// TwinCAT 3 PLC project PLC
// ProgramVersion: 3.1.4026.16
// libraries:
//   Tc2_ModbusRTU, * (Beckhoff Automation GmbH)
//   Tc2_Standard, * (Beckhoff Automation GmbH)
//   Tc2_SUPS, * (Beckhoff Automation GmbH)
//   Tc2_System, * (Beckhoff Automation GmbH)
//   Tc2_Utilities, * (Beckhoff Automation GmbH)
//   Tc3_Database, * (Beckhoff Automation GmbH)
//   Tc3_EventLogger, * (Beckhoff Automation GmbH)
// project tree:
//   DUTs/Database/ ST_AuditTrail.TcDUT, ST_BatchData.TcDUT, ST_OperatorAct.TcDUT, ST_ProcessData.TcDUT
//   DUTs/ EN_BatchEvents.TcDUT, EN_RecipeType.TcDUT, ST_Alarm.TcDUT, ST_Batch.TcDUT, ST_Control.TcDUT, ST_Diagnostic.TcDUT, ST_HMI.TcDUT, ST_HMI_Time.TcDUT, ST_LastBatch.TcDUT, ST_OPC.TcDUT, ST_ProcessCmd.TcDUT, ST_PythonHandshake.TcDUT, ST_RecipeList.TcDUT, ST_Report.TcDUT, ST_RX_Python.TcDUT, ST_Settings.TcDUT, ST_Time.TcDUT, ST_ToHMI.TcDUT, ST_TONP.TcDUT, ST_TX_Python.TcDUT
//   DUTs/Recipe/ ST_Cleaning_Phases.TcDUT, ST_Production_Phases.TcDUT, ST_Recipe_Production.TcDUT, ST_RecipeInfo.TcDUT, ST_Recipe_Cleaning.TcDUT
//   DUTs/ST_HMI/ ST_AlarmControl.TcDUT, ST_AuditControl.TcDUT, ST_BatchControl.TcDUT, ST_MachineControl.TcDUT, ST_ProcessControl.TcDUT, ST_RecipeControl.TcDUT, ST_ReportControl.TcDUT
//   DUTs/ST_ToHMI/ ST_Devices.TcDUT, ST_EnableControls.TcDUT, ST_Pipes.TcDUT, ST_ProcessVar.TcDUT, ST_Status.TcDUT
//   FB/Database/ FB_WriteChange.TcPOU, FB_WriteChange_STR.TcPOU, FB_WriteClick.TcPOU, FB_WriteEvent.TcPOU
//   FB/ FB_AnalogOutput.TcPOU, FB_AVG200.TcPOU, FB_Batch.TcPOU, FB_BatchLog.TcPOU, FB_Chopper_Ctrl.TcPOU, FB_Coil_Ctrl.TcPOU, FB_DeleteOldestFile.TcPOU, FB_FileSaveAs.TcPOU, FB_FileSaveAs_V02.TcPOU, FB_Mixer_Ctrl.TcPOU, FB_PythonScript.TcPOU, FB_Scale.TcPOU, FB_SystemDateTime.TcPOU, FB_TimeElapsed_HMI.TcPOU, FB_TONP.TcPOU, FB_Valve53_Ctrl.TcPOU, FB_Valve_Ctrl.TcPOU, F_Interlocks.TcPOU, F_OperationalTime.TcPOU, F_StepCMP.TcPOU, F_TimeBarHMI.TcPOU, F_TimerHMI.TcPOU
//   GVLs/ CONST.TcGVL, GV.TcGVL, IN.TcGVL, OUT.TcGVL, Recipes.TcGVL
//   Mapping/ ST_EL1819.TcDUT, ST_EL2809.TcDUT, ST_EL3174.TcDUT, ST_EL3214.TcDUT, ST_EL4008.TcDUT, ST_EL4124.TcDUT, ST_EL6021.TcDUT, ST_EL9110.TcDUT
//   / PlcTask.TcTTO
//   POUs/1. Main Control/ P1_00_MAIN.TcPOU, P1_01_Recipe.TcPOU, P1_02_Batch.TcPOU, P1_04_MachineControl.TcPOU, P1_03_Alarms.TcPOU
//   POUs/2. Process/Cleaning/ _Blowing.TcPOU, _Control.TcPOU, _Draining.TcPOU, _MainClean.TcPOU, _Mounting.TcPOU, _PreWash.TcPOU
//   POUs/2. Process/ P2_00_MAIN.TcPOU, P2_01_Production_Seq.TcPOU, P2_02_Cleaning_Seq.TcPOU, P2_03_Production_Ctrl.TcPOU, P2_04_Cleaning_Ctrl.TcPOU, P2_05_Process_Ctrl.TcPOU, P2_06_Device_Ctrl.TcPOU, _Chopper.TcPOU, _Mixer.TcPOU
//   POUs/2. Process/Production/ _Discharging.TcPOU, _Feeding.TcPOU, _Mixing.TcPOU
//   POUs/3. Report/ P3_00_MAIN.TcPOU, P3_01_BatchData.TcPOU, P3_03_ProcessData.TcPOU, P3_04_Alarms.TcPOU, P3_06_CreateReport.TcPOU, P3_07_SendReport.TcPOU, P3_08_OpenReport.TcPOU
//   POUs/4. Audit Trail/ P4_00_MAIN.TcPOU, P4_01_Write.TcPOU, P4_02_Read.TcPOU, P4_03_Export.TcPOU, P4_04_Delete.TcPOU, P4_05_DIskSize.TcPOU, P4_05_Send.TcPOU
//   POUs/5. HMI/ P5_00_MAIN.TcPOU, P5_01_EnableControls.TcPOU, P5_02_DiagramVisualisation.TcPOU, P5_03_OtherControl.TcPOU, P5_04_BatchStatus.TcPOU, P5_05_Screenshot.TcPOU, P5_06_Trends.TcPOU
//   POUs/ MAIN.TcPOU, P00_Mapping.TcPOU, P01_AnalogScaling.TcPOU, P02_GlobalSystemTime.TcPOU
// real-time tasks:
//   TASK PlcTask: cycle T#10ms, priority 20, ADS port 350
// I/O:
//   DEVICE PLC-ECAT (disabled), AmsNetId 169.254.227.12.5.1
//     BUS-ETCAT [EK1100 EtherCAT Coupler (2A E-Bus)]
//       PT100 (EL3214) (EL3214) [EL3214 4Ch. Ana. Input PT100 (RTD)]
//       Analog Input #1 (EL3174) [EL3174 4Ch. Ana. Input +/-10V Diff., +/-20mA SingleEnded, 16 Bit]
//       Analog Input #2 (EL3174) [EL3174 4Ch. Ana. Input +/-10V Diff., +/-20mA SingleEnded, 16 Bit]
//       Digital Input #1 (EL1819) [EL1819 16Ch. Dig. Input 24V, 10µs]
//       Analog Output #1 (EL4008) [EL4008 8Ch. Ana. Output 0-10V, 12bit]
//       Power Supply (EL9110) [EL9110 Power Supplier with LED (24V, Diagnostics)]
//       Digital Output #1 (EL2809) [EL2809 16Ch. Dig. Output 24V, 0.5A]
//       Digital Output #2 (EL2809) [EL2809 16Ch. Dig. Output 24V, 0.5A]
//       Modbus (EL6021) [EL6021 Interface (RS422/485)]
//       Term 9 (EL9011) [EL9011 End Terminal]
// variable links:
//   (this object) <-> PLC-ECAT/BUS-ETCAT/Analog Input #1 (EL3174)
//     PlcTask Inputs/P00_Mapping.AI1.Ch1_Error <-> AI Standard Channel 1/Status/Error
//     PlcTask Inputs/P00_Mapping.AI1.Ch2_Error <-> AI Standard Channel 2/Status/Error
//     PlcTask Inputs/P00_Mapping.AI1.Ch3_Error <-> AI Standard Channel 3/Status/Error
//     PlcTask Inputs/P00_Mapping.AI1.Ch4_Error <-> AI Standard Channel 4/Status/Error
//     PlcTask Inputs/P00_Mapping.AI1.Ch1_Value <-> AI Standard Channel 1/Value
//     PlcTask Inputs/P00_Mapping.AI1.Ch2_Value <-> AI Standard Channel 2/Value
//     PlcTask Inputs/P00_Mapping.AI1.Ch3_Value <-> AI Standard Channel 3/Value
//     PlcTask Inputs/P00_Mapping.AI1.Ch4_Value <-> AI Standard Channel 4/Value
//     PlcTask Inputs/P00_Mapping.AI1.State <-> InfoData/State
//   (this object) <-> PLC-ECAT/BUS-ETCAT/Analog Input #2 (EL3174)
//     PlcTask Inputs/P00_Mapping.AI2.Ch1_Error <-> AI Standard Channel 1/Status/Error
//     PlcTask Inputs/P00_Mapping.AI2.Ch2_Error <-> AI Standard Channel 2/Status/Error
//     PlcTask Inputs/P00_Mapping.AI2.Ch3_Error <-> AI Standard Channel 3/Status/Error
//     PlcTask Inputs/P00_Mapping.AI2.Ch4_Error <-> AI Standard Channel 4/Status/Error
//     PlcTask Inputs/P00_Mapping.AI2.Ch1_Value <-> AI Standard Channel 1/Value
//     PlcTask Inputs/P00_Mapping.AI2.Ch2_Value <-> AI Standard Channel 2/Value
//     PlcTask Inputs/P00_Mapping.AI2.Ch3_Value <-> AI Standard Channel 3/Value
//     PlcTask Inputs/P00_Mapping.AI2.Ch4_Value <-> AI Standard Channel 4/Value
//     PlcTask Inputs/P00_Mapping.AI2.State <-> InfoData/State
//   (this object) <-> PLC-ECAT/BUS-ETCAT/Analog Output #1 (EL4008)
//     PlcTask Inputs/P00_Mapping.AO1.State <-> InfoData/State
//     PlcTask Outputs/P00_Mapping.AO1.Ch1_Value <-> AO Outputs Channel 1/Analog output
//     PlcTask Outputs/P00_Mapping.AO1.Ch2_Value <-> AO Outputs Channel 2/Analog output
//     PlcTask Outputs/P00_Mapping.AO1.Ch3_Value <-> AO Outputs Channel 3/Analog output
//     PlcTask Outputs/P00_Mapping.AO1.Ch4_Value <-> AO Outputs Channel 4/Analog output
//   (this object) <-> PLC-ECAT/BUS-ETCAT/Digital Input #1 (EL1819)
//     PlcTask Inputs/P00_Mapping.DI1.Ch10_Value <-> Channel 10/Input
//     PlcTask Inputs/P00_Mapping.DI1.Ch11_Value <-> Channel 11/Input
//     PlcTask Inputs/P00_Mapping.DI1.Ch12_Value <-> Channel 12/Input
//     PlcTask Inputs/P00_Mapping.DI1.Ch13_Value <-> Channel 13/Input
//     PlcTask Inputs/P00_Mapping.DI1.Ch14_Value <-> Channel 14/Input
//     PlcTask Inputs/P00_Mapping.DI1.Ch15_Value <-> Channel 15/Input
//     PlcTask Inputs/P00_Mapping.DI1.Ch16_Value <-> Channel 16/Input
//     PlcTask Inputs/P00_Mapping.DI1.Ch1_Value <-> Channel 1/Input
//     PlcTask Inputs/P00_Mapping.DI1.Ch2_Value <-> Channel 2/Input
//     PlcTask Inputs/P00_Mapping.DI1.Ch3_Value <-> Channel 3/Input
//     PlcTask Inputs/P00_Mapping.DI1.Ch4_Value <-> Channel 4/Input
//     PlcTask Inputs/P00_Mapping.DI1.Ch5_Value <-> Channel 5/Input
//     PlcTask Inputs/P00_Mapping.DI1.Ch6_Value <-> Channel 6/Input
//     PlcTask Inputs/P00_Mapping.DI1.Ch7_Value <-> Channel 7/Input
//     PlcTask Inputs/P00_Mapping.DI1.Ch8_Value <-> Channel 8/Input
//     PlcTask Inputs/P00_Mapping.DI1.Ch9_Value <-> Channel 9/Input
//     PlcTask Inputs/P00_Mapping.DI1.State <-> InfoData/State
//   (this object) <-> PLC-ECAT/BUS-ETCAT/Digital Output #1 (EL2809)
//     PlcTask Inputs/P00_Mapping.DO1.State <-> InfoData/State
//     PlcTask Outputs/P00_Mapping.DO1.Ch10_Value <-> Channel 10/Output
//     PlcTask Outputs/P00_Mapping.DO1.Ch11_Value <-> Channel 11/Output
//     PlcTask Outputs/P00_Mapping.DO1.Ch12_Value <-> Channel 12/Output
//     PlcTask Outputs/P00_Mapping.DO1.Ch13_Value <-> Channel 13/Output
//     PlcTask Outputs/P00_Mapping.DO1.Ch14_Value <-> Channel 14/Output
//     PlcTask Outputs/P00_Mapping.DO1.Ch15_Value <-> Channel 15/Output
//     PlcTask Outputs/P00_Mapping.DO1.Ch16_Value <-> Channel 16/Output
//     PlcTask Outputs/P00_Mapping.DO1.Ch1_Value <-> Channel 1/Output
//     PlcTask Outputs/P00_Mapping.DO1.Ch2_Value <-> Channel 2/Output
//     PlcTask Outputs/P00_Mapping.DO1.Ch3_Value <-> Channel 3/Output
//     PlcTask Outputs/P00_Mapping.DO1.Ch4_Value <-> Channel 4/Output
//     PlcTask Outputs/P00_Mapping.DO1.Ch5_Value <-> Channel 5/Output
//     PlcTask Outputs/P00_Mapping.DO1.Ch6_Value <-> Channel 6/Output
//     PlcTask Outputs/P00_Mapping.DO1.Ch7_Value <-> Channel 7/Output
//     PlcTask Outputs/P00_Mapping.DO1.Ch8_Value <-> Channel 8/Output
//     PlcTask Outputs/P00_Mapping.DO1.Ch9_Value <-> Channel 9/Output
//   (this object) <-> PLC-ECAT/BUS-ETCAT/Digital Output #2 (EL2809)
//     PlcTask Inputs/P00_Mapping.DO2.State <-> InfoData/State
//     PlcTask Outputs/P00_Mapping.DO2.Ch10_Value <-> Channel 10/Output
//     PlcTask Outputs/P00_Mapping.DO2.Ch11_Value <-> Channel 11/Output
//     PlcTask Outputs/P00_Mapping.DO2.Ch12_Value <-> Channel 12/Output
//     PlcTask Outputs/P00_Mapping.DO2.Ch13_Value <-> Channel 13/Output
//     PlcTask Outputs/P00_Mapping.DO2.Ch14_Value <-> Channel 14/Output
//     PlcTask Outputs/P00_Mapping.DO2.Ch15_Value <-> Channel 15/Output
//     PlcTask Outputs/P00_Mapping.DO2.Ch16_Value <-> Channel 16/Output
//     PlcTask Outputs/P00_Mapping.DO2.Ch1_Value <-> Channel 1/Output
//     PlcTask Outputs/P00_Mapping.DO2.Ch2_Value <-> Channel 2/Output
//     PlcTask Outputs/P00_Mapping.DO2.Ch3_Value <-> Channel 3/Output
//     PlcTask Outputs/P00_Mapping.DO2.Ch4_Value <-> Channel 4/Output
//     PlcTask Outputs/P00_Mapping.DO2.Ch5_Value <-> Channel 5/Output
//     PlcTask Outputs/P00_Mapping.DO2.Ch6_Value <-> Channel 6/Output
//     PlcTask Outputs/P00_Mapping.DO2.Ch7_Value <-> Channel 7/Output
//     PlcTask Outputs/P00_Mapping.DO2.Ch8_Value <-> Channel 8/Output
//     PlcTask Outputs/P00_Mapping.DO2.Ch9_Value <-> Channel 9/Output
//   (this object) <-> PLC-ECAT/BUS-ETCAT/Modbus (EL6021)
//     PlcTask Inputs/P00_Mapping.PB1.State <-> COM TxPDO-Map Inputs/Status
//   (this object) <-> PLC-ECAT/BUS-ETCAT/PT100 (EL3214) (EL3214)
//     PlcTask Inputs/P00_Mapping.TI1.Ch1_Error <-> RTD Inputs Channel 1/Status/Error
//     PlcTask Inputs/P00_Mapping.TI1.Ch2_Error <-> RTD Inputs Channel 2/Status/Error
//     PlcTask Inputs/P00_Mapping.TI1.Ch3_Error <-> RTD Inputs Channel 3/Status/Error
//     PlcTask Inputs/P00_Mapping.TI1.Ch4_Error <-> RTD Inputs Channel 4/Status/Error
//     PlcTask Inputs/P00_Mapping.TI1.Ch1_Value <-> RTD Inputs Channel 1/Value
//     PlcTask Inputs/P00_Mapping.TI1.Ch2_Value <-> RTD Inputs Channel 2/Value
//     PlcTask Inputs/P00_Mapping.TI1.Ch3_Value <-> RTD Inputs Channel 3/Value
//     PlcTask Inputs/P00_Mapping.TI1.Ch4_Value <-> RTD Inputs Channel 4/Value
//     PlcTask Inputs/P00_Mapping.TI1.State <-> InfoData/State
//   (this object) <-> PLC-ECAT/BUS-ETCAT/Power Supply (EL9110)
//     PlcTask Inputs/P00_Mapping.PS1.PowerOK <-> PowerOK/Input
//     PlcTask Inputs/P00_Mapping.PS1.State <-> InfoData/State

CONFIGURATION PLC
    RESOURCE PLC ON TwinCAT3
        TASK PlcTask(INTERVAL := T#10ms, PRIORITY := 20);
        PROGRAM MAIN WITH PlcTask : MAIN;
    END_RESOURCE
END_CONFIGURATION

// ---- DUTs/Database/ST_AuditTrail.TcDUT
TYPE ST_AuditTrail :
STRUCT
	DateTime	: DT;
	User		: STRING(100);
	Event		: STRING(100);
	Description	: STRING(100);
	Oldvalue	: STRING(100);
	Newvalue	: STRING(100);	
END_STRUCT
END_TYPE

// ---- DUTs/Database/ST_BatchData.TcDUT
TYPE ST_BatchData :
STRUCT
	Batch		: STRING(100);
	Parameter	: STRING(100);
	Value		: STRING(100);
END_STRUCT
END_TYPE

// ---- DUTs/Database/ST_OperatorAct.TcDUT
TYPE ST_OperatorAct :
STRUCT
	Batch		: STRING(100);
	DateTime	: DT;
	Event		: STRING(100);
	Description	: STRING(100);
END_STRUCT
END_TYPE

// ---- DUTs/Database/ST_ProcessData.TcDUT
TYPE ST_ProcessData :
STRUCT
	Batch		: STRING(100);
	DateTime	: DT;
	Value1		: STRING(100);
	Value2		: STRING(100);
	Value3		: STRING(100);
	Value4		: STRING(100);
	Value5		: STRING(100);
	Value6		: STRING(100);
	Value7		: STRING(100);
END_STRUCT
END_TYPE

// ---- DUTs/EN_BatchEvents.TcDUT
{attribute 'to_string'}
TYPE EN_BatchEvents :
(
	ALL				:= 0,
	RECIPE		    := 1,
	BATCH			:= 2,
	SETTINGS		:= 3,
	CALIBRATION		:= 4,
	ACTIONS			:= 5
);
END_TYPE

// ---- DUTs/EN_RecipeType.TcDUT
{attribute 'to_string'}
TYPE EN_RecipeType :
(
	Production			:= 0,
	Cleaning		    := 1
);
END_TYPE

// ---- DUTs/Recipe/ST_Cleaning_Phases.TcDUT
TYPE ST_Cleaning_Phases :
STRUCT
	bEnable								:BOOL;
	iType								:INT;  //0-Prewash,1- Filter-Dismout-Nozzle-Mount, 2-Main Clean, 3 - PW Clean, 4 - Rinising pipes, 5 Blowing out, 6 - Control
	sDescription						:STRING;
	rMixingShaft_Speed					:REAL;
	iMixer								:INT;  //0-OFF,1-ON/Forward,2-Interval,3-Backward,4-Alternate
	iChopper							:INT;  //0-OFF,1-ON
	iMedium								:INT;  //0-Cold water,1-Warm water,2-Purified water
	iDetergent							:INT;  //0-OFF,1-ON
	iTime1								:ST_HMI_Time;			
	iTime2								:ST_HMI_Time;
	iTime3								:ST_HMI_Time;
END_STRUCT
END_TYPE

// ---- DUTs/Recipe/ST_Production_Phases.TcDUT
TYPE ST_Production_Phases :
STRUCT
	bEnable					:BOOL;
	iType					:INT;  	//0-Feeding,1-Mixing,2-Discharging
	sDescription			:STRING;
	iEndPoint				:INT;    //0-Manual,1-Auto
	iPhaseTime				:ST_HMI_Time;
	iMixing					:INT; 	//0-OFF,1-ON/Forward,2-Interval,3-Backward,4-Alternate
	rMixingShaft_Speed		:REAL;
	iChopper				:INT;	//0-OFF,1-Slow,2-Fast
END_STRUCT
END_TYPE

// ---- DUTs/Recipe/ST_Recipe_Production.TcDUT
TYPE ST_Recipe_Production :
STRUCT
	sName					:STRING[80];
	stInfo					:ST_RecipeInfo;
	stPhase					:ARRAY[0..20] OF ST_Production_Phases;
	iType					:INT; 
	iActivePhase			:INT;
END_STRUCT
END_TYPE

// ---- DUTs/Recipe/ST_RecipeInfo.TcDUT
TYPE ST_RecipeInfo :
STRUCT
	sUserCreated		:STRING;
	sUserEdited			:STRING;
	sUserVerified		:STRING;
	sTimeCreated		:STRING;
	sTimeEdited			:STRING;
	sTimeVerified		:STRING;
	bVerification		:BOOL;
	iVersion			:INT;
END_STRUCT
END_TYPE

// ---- DUTs/Recipe/ST_Recipe_Cleaning.TcDUT
TYPE ST_Recipe_Cleaning :
STRUCT
	sName					:STRING[80];
	stInfo					:ST_RecipeInfo;
	stPhase					:ARRAY[0..20] OF ST_Cleaning_Phases;
	iType					:INT; 
	iActivePhase			:INT;
END_STRUCT
END_TYPE

// ---- DUTs/ST_Alarm.TcDUT
TYPE ST_Alarm :
STRUCT
	Alarm			:ARRAY[0..99] OF fb_TcAlarm;
	Active			:ARRAY[0..99] OF BOOL;
	Raise			:ARRAY[0..99] OF BOOL;
	
	Warning			:ARRAY[0..99] OF fb_TcAlarm;
	Message			:ARRAY[0..99] OF BOOL;
	
END_STRUCT
END_TYPE

// ---- DUTs/ST_Batch.TcDUT
TYPE ST_Batch :
STRUCT
	sBatchNumber		:STRING;
	sBatchName			:STRING;
	sRecipeName			:STRING;
	sRecipeType			:STRING;
	sProductName		:STRING;
	sComment			:STRING;
	sUser				:STRING;
	sStarted			:STRING;
	sFinished			:STRING;
END_STRUCT
END_TYPE

// ---- DUTs/ST_Control.TcDUT
TYPE ST_Control :
STRUCT
	Auto				:BOOL;
	Manual				:BOOL;
	Maintenance			:BOOL;
	
	Starting			:BOOL;
	Running				:BOOL;
	Stop				:BOOL;
	Stopping			:BOOL;
	Paused				:BOOL;
	Stopped				:BOOL;
	Finish				:BOOL;
	
	Next				:BOOL;
	Previous			:BOOL;
	Jump				:BOOL;
	JumpStep			:INT;
	
	Recovery			:BOOL;
	Confirmation		:BOOL;
	Operation			:BOOL;
	
	Intelrocks			:BOOL;
	Processlocks		:BOOL;
	
END_STRUCT
END_TYPE

// ---- DUTs/ST_Diagnostic.TcDUT
TYPE ST_Diagnostic :
STRUCT
	Temperature			:UDINT;
	BootCount			:UDINT;
	OperationTime		:UDINT;
	OperationDuration	:ARRAY[0..2] OF INT;
END_STRUCT
END_TYPE

// ---- DUTs/ST_HMI.TcDUT
TYPE ST_HMI :
STRUCT
		stBatch_Ctrl						:ST_BatchControl;
		stRecipeProd_Ctrl					:ST_RecipeControl;
		stRecipeClean_Ctrl					:ST_RecipeControl;
		stMachine_Ctrl						:ST_MachineControl;
		stAlarm_Ctrl						:ST_AlarmControl;
		stAudit_Ctrl						:ST_AuditControl;
		stReport_Ctrl						:ST_ReportControl;
		stProcess_Ctrl						:ST_ProcessControl;
		
		stRecipeProd						:ST_Production_Phases;
		stRecipeClean						:ST_Cleaning_Phases;
		
		stActiveRecipeProd					:ST_Production_Phases;
		stActiveRecipeClean					:ST_Cleaning_Phases;
		
		bScreenShot							:BOOL;
		bCloseApp							:BOOL;
		
		
		bUserLogIn							:BOOL;
		bUserLogOut							:BOOL;
		bStayLoggedIn						:BOOL;
		
		iStepTime1Prod_RectWidth			:INT;
		iStepTime1_RectWidth				:INT;
		iStepTime2_RectWidth				:INT;
		iStepTime3_RectWidth				:INT;
		iStepTime4_RectWidth				:INT;
		iStepTime5_RectWidth				:INT;
		iStepTime6_RectWidth				:INT;
		iStepTime7_RectWidth				:INT;
		
END_STRUCT
END_TYPE

// ---- DUTs/ST_HMI/ST_AlarmControl.TcDUT
TYPE ST_AlarmControl :
STRUCT
	bAckAll					:BOOL;
	bFilter					:BOOL;
END_STRUCT
END_TYPE

// ---- DUTs/ST_HMI/ST_AuditControl.TcDUT
TYPE ST_AuditControl :
STRUCT
	bReadDB							:BOOL;
	bReadDBSize						:BOOL;

	bFilter							:BOOL;
	bClear							:BOOL;
	sFilter_Key						:STRING;
	dtFilter_From					:DT;
	dtFilter_To						:DT;
	sFilter_User					:STRING;
	enFilter_Event					:EN_BatchEvents;
	iViewFilter						:BOOL;
	
	bExport							:BOOL;
	sExportName						:STRING;
	
	bDelete							:BOOL;
	bSend							:BOOL;
	
	iProdSelectedProcess			:INT;
	iCleanSelectedProcess			:INT;
	iBatchSelectedProcess			:INT;
	
	bScanRecipeParams				:BOOL;
	bScanPhases						:BOOL;
END_STRUCT
END_TYPE

// ---- DUTs/ST_HMI/ST_BatchControl.TcDUT
TYPE ST_BatchControl :
STRUCT
	bCreate			:BOOL;
	bCancel			:BOOL;
	bOpen			:BOOL;
	bClose			:BOOL;
	bLoad			:BOOL;
	
	sName			:STRING;
	iNumber			:UDINT;
	sProduct		:STRING;
	sComment		:STRING;
	sRecipe			:STRING;
	
	iRecipeType		:INT;
END_STRUCT
END_TYPE

// ---- DUTs/ST_HMI/ST_MachineControl.TcDUT
TYPE ST_MachineControl :
STRUCT
	bAuto					:BOOL;
	bManual					:BOOL;
	bMaintenance			:BOOL;
	bStart					:BOOL;
	bStop					:BOOL;
	bPause					:BOOL;
	bDoorClose				:BOOL;	
	bDoorOpen				:BOOL;
	bNext					:BOOL;
	bPrevious				:BOOL;
END_STRUCT
END_TYPE

// ---- DUTs/ST_HMI/ST_ProcessControl.TcDUT
TYPE ST_ProcessControl :
STRUCT

	bVacuumPump					:BOOL;
	bFinishFeeding				:BOOL;
	bEnableMixer				:BOOL;
	bBarrelInPos				:BOOL;
	bFinishDischarge			:BOOL;
	bFinishDetergent			:BOOL;
	bFinishMixing				:BOOL;
	bFinishMounting				:BOOL;
	bFinishControlOK			:BOOL;
	bFinishControlNOK			:BOOL;
	
	
	bBatchConfirm1				:BOOL;
	bBatchConfirm2				:BOOL;
	bBatchConfirm3				:BOOL;
	bBatchConfirm4				:BOOL;
	
	bDischargeFlap_Open			:BOOL;
	bDischargeFlap_HOpen		:BOOL;
	bDischargeFlap_Close		:BOOL;
	
	bBlowing					:BOOL;
END_STRUCT
END_TYPE

// ---- DUTs/ST_HMI/ST_RecipeControl.TcDUT
TYPE ST_RecipeControl :
STRUCT
	iType					:INT;
	bCreate					:BOOL;
	bRefresh				:BOOL;
	bOpen					:BOOL;
	bClose					:BOOL;
	bDelete					:BOOL;
	iIndex					:INT;
	iList					:INT;
END_STRUCT
END_TYPE

// ---- DUTs/ST_HMI/ST_ReportControl.TcDUT
TYPE ST_ReportControl :
STRUCT
	iIndex					:INT;
END_STRUCT
END_TYPE

// ---- DUTs/ST_HMI_Time.TcDUT
TYPE ST_HMI_Time :
STRUCT
	mins				:DINT; 		//Minutes
	sec					:DINT; 		//Seconds
END_STRUCT
END_TYPE

// ---- DUTs/ST_LastBatch.TcDUT
TYPE ST_LastBatch :
STRUCT
	iType					:INT;
	sBatchNumber			:STRING;
	sRecipe					:STRING;
	sUser					:STRING;
	sStarted				:STRING;
	sFinished				:STRING;

END_STRUCT
END_TYPE

// ---- DUTs/ST_OPC.TcDUT
TYPE ST_OPC :
STRUCT
	BatchType				:STRING;
	BatchTime				:DINT;
	BatchID					:STRING;
	PhaseName				:STRING;
	RecipeName				:STRING;
	PhaseTime				:DINT;
	MixerActualSpeed		:REAL;
	MixerMaxSpeed			:REAL;
	ChopperCommand			:BOOL;
	Temperature				:REAL;
	MachineStatus			:STRING;
	sMixingStartTime		:STRING;
	sMixingStopTime			:STRING;
	sMixingSetpoint			:DINT;
	
END_STRUCT
END_TYPE

// ---- DUTs/ST_ProcessCmd.TcDUT
TYPE ST_ProcessCmd :
STRUCT
	iMixer					:INT;
	rMixerSpeed				:REAL;
	iChopper				:INT;
	
	bMixerFwd				:BOOL;
	bMixerBcw				:BOOL;
	bChopper				:BOOL;
	
	bDryingSocketPipe		:BOOL;
	
	bWater					:BOOL;
	bWarmWater				:BOOL;
	bColdWater				:BOOL;
	bProcessWater			:BOOL;
	bAir					:BOOL;
	
	bTightAir				:BOOL;
	
	bChopper1_Air			:BOOL;
	bChopper1_Water			:BOOL;
	bChopper1_Drain			:BOOL;
		
	bChopper2_Air			:BOOL;
	bChopper2_Water			:BOOL;
	bChopper2_Drain			:BOOL;
		
	
	bDischargeOpen			:BOOL;
	bDischargeClose			:BOOL;
	bDischargeHalfOpen		:BOOL;
	bDischargeFix			:BOOL;
	
END_STRUCT
END_TYPE

// ---- DUTs/ST_PythonHandshake.TcDUT
TYPE ST_PythonHandshake :
STRUCT
	bBusy					:BOOL;
	bDone					:BOOL;
	bError					:BOOL;
	sError					:STRING(255);
END_STRUCT
END_TYPE

// ---- DUTs/ST_RecipeList.TcDUT
TYPE ST_RecipeList :
STRUCT
	sName			:STRING;
	sCreated		:STRING;
	sEdited			:STRING;
	sVerified		:STRING[3];
END_STRUCT
END_TYPE

// ---- DUTs/ST_Report.TcDUT
TYPE ST_Report :
STRUCT
	bStartCreate_Sequence				:BOOL;
	bStartSend_Sequence					:BOOL;
	bSend_Report						:BOOL;
	bExport_Alarms						:BOOL;
	bSaveAs_Alarms						:BOOL;
	bCreate_Report						:BOOL;
	bDelete_Data						:BOOL;
	bDelete_OldestReport				:BOOL;
END_STRUCT
END_TYPE

// ---- DUTs/ST_RX_Python.TcDUT
TYPE ST_RX_Python :
STRUCT
	stAuditExport				:ST_PythonHandshake;
	stSendReport				:ST_PythonHandshake;
	stBatchReport				:ST_PythonHandshake;
	stDiskCapacity				:ST_PythonHandshake;
	sDiskFree					:STRING(255);
	sDisckCapacity				:STRING(255);
END_STRUCT
END_TYPE

// ---- DUTs/ST_Settings.TcDUT
TYPE ST_Settings :
STRUCT
	iReportProcesData_TimeStamp		:DINT;
	iMixerInterval_Run_sec			:DINT;
	iMixerInterval_Pause_sec		:DINT;
	iMixerAlternate_Run_sec			:DINT;
	iMixerAlternate_Pause_sec		:DINT;
	iAutoLogOutTimeOut_min			:DINT;
	rProductTemperature_Offset		:REAL;
	
	rMixerL_Flow_ThresholdMin		:REAL;
	rMixerR_Flow_ThresholdMin		:REAL;
	rChopper1_Flow_ThresholdMin		:REAL;
	rChopper2_Flow_ThresholdMin		:REAL;
	
	rMixerL_Flow_ThresholdMax		:REAL;
	rMixerR_Flow_ThresholdMax		:REAL;
	rChopper1_Flow_ThresholdMax		:REAL;
	rChopper2_Flow_ThresholdMax		:REAL;
	
	bDischargeFlap_Manual			:BOOL;
	iDischargeFlap_TimeOut			:DINT;
	iDischargeFlapHalf_TimeOut		:DINT;
	
	rMixerDischargeSpeed			:REAL;
	iBlowingChopperCmd				:INT;
	iBlowingMixerCmd				:INT;
	rBlowingMixerSpeed				:REAL;
	iFillingChopperOnTime			:DINT;
END_STRUCT
END_TYPE

// ---- DUTs/ST_Time.TcDUT
TYPE ST_Time :
STRUCT
	dtDateTime			:DT;
	sTime				:STRING;
	sDate				:STRING;
	sDateTime			:STRING;
	sFormatDateTime		:STRING;
	bClock_500ms		:BOOL;
	bClock_1s			:BOOL;
	bClock_2s			:BOOL;
	bClock_5s			:BOOL;
	bClock_60s			:BOOL;
	bClock_1OFF_2ON		:BOOL;
	bPulse_10s			:BOOL;
	bPulse_30s			:BOOL;
	bPulse_60s			:BOOL;
	bCustomBlink1		:BOOL;
	bCustomBlink2		:BOOL;
	bCustomBlink3		:BOOL;
	bNewDay				:BOOL;
	bNewMonth			:BOOL;
	bNewYear			:BOOL;
END_STRUCT
END_TYPE

// ---- DUTs/ST_ToHMI.TcDUT
TYPE ST_ToHMI :
STRUCT
	stControlsEN				:ST_EnableControls;
	stPipes						:ST_Pipes;
	stDevices					:ST_Devices;
	stStatus					:ST_Status;
	stProcessVar				:ST_ProcessVar;
	iRecipeProd_Number			:INT;
	iRecipeClean_Number			:INT;
	sReporth_OpenPath			:STRING;
	sAudit_OpenPath				:STRING;
	sUserMan_OpenPath			:STRING;
	iBatchStep					:INT;
	
	sUserLogged					:STRING;
	sActiveBatch				:STRING;
	sActiveRecipe				:STRING;
	bBatchOpen					:BOOL;
	
	sMixingTime_VIS				:STRING;
	sMixingDone_VIS				:STRING;
	bDetergentConfirm_VIS		:BOOL;
	bDischargeConfirm_VIS		:BOOL;
	
	bAlarm						:BOOL;
	bAlarm_Blink				:BOOL;
	
	bUserTimeOut				:BOOL;
	bUserLogOut					:BOOL;
	bLogInDefaultUser			:BOOL;
	
	
END_STRUCT
END_TYPE

// ---- DUTs/ST_ToHMI/ST_Devices.TcDUT
TYPE ST_Devices :
STRUCT
	iMixer					:INT; 		//0-OFF, 1-Forward Slow, 2-Forward Fast, 3-Backward Slow, 4-Backward Fast
	iChopper1				:INT;		//0-OFF, 1-ON
	iChopper2				:INT;		//0-OFF, 1-ON
	iHeater					:INT;
	bFlowMixerL_OK			:BOOL;
	bFlowMixerR_OK			:BOOL;
	bFlowChopper1_OK		:BOOL;
	bFlowChopper2_OK		:BOOL;
	bDoorClosed				:BOOL;
	bDoorReadyToLock		:BOOL;
	bDischargeFlap			:BOOL;
END_STRUCT
END_TYPE

// ---- DUTs/ST_ToHMI/ST_EnableControls.TcDUT
TYPE ST_EnableControls :
STRUCT
	bAuto_Button				:BOOL;
	bManual_Button				:BOOL;
	bMaintenance_Button			:BOOL;
	bStart_Button				:BOOL;
	bStop_Button				:BOOL;
	bPause_Button				:BOOL;
	bNext_Button				:BOOL;
	bPrevious_Button			:BOOL;
	bDoorLock_Button			:BOOL;
	bDoorUnlock_Button			:BOOL;
	bVacuum_Button				:BOOL;
	bMixer_Button				:BOOL;
	bBatchCreate_Button			:BOOL;
	bScreenShot_Img				:BOOL;
	bDischargeOpen_Button		:BOOL;
	bDIschargeClose_Button		:BOOL;
	bBlowing_Button				:BOOL;
	bRecipeCreate_Button		:BOOL;
END_STRUCT
END_TYPE

// ---- DUTs/ST_ToHMI/ST_Pipes.TcDUT
TYPE ST_Pipes :
STRUCT
	
	//0-OFF, 1-Air Blow, 2-Cold Water(PW), 3-Warm water, 4 - PW						


	iWaterSupply							:INT; 	
	iColdWater								:INT;
	iWarmWater								:INT;
	iWaterSelect							:INT;
	iProcessWater							:INT;
	iMainSupply								:INT;
	iTightAir								:INT;
	iChopper1								:INT;
	iChopper2								:INT;
	iChopper1Drain							:INT;
	iChopper2Drain							:INT;
	iChoppersDrain							:INT;
	iMainDrain								:INT;	
	iAirBlow								:INT;
	iChopper1Air							:INT;
	iChopper2Air							:INT;	

	//0-OFF,1-Production OFF,2-Production ON,3-Cleaning OFF,4 Clening ON
	iFluid									:INT;		
END_STRUCT
END_TYPE

// ---- DUTs/ST_ToHMI/ST_ProcessVar.TcDUT
TYPE ST_ProcessVar :
STRUCT
	rMixerSpeed					:REAL;
	rMixerCurrent				:REAL;
	rChopper1Current			:REAL;
	rChopper2Current			:REAL;
	rProductTemperature			:REAL;
	rFlowChopper1				:REAL;
	rFlowChopper2				:REAL;
	rFlowMixerL					:REAL;
	rFlowMixerR					:REAL;
END_STRUCT
END_TYPE

// ---- DUTs/ST_ToHMI/ST_Status.TcDUT
TYPE ST_Status :
STRUCT
	sBatchTime							:STRING; 	//Time elapsed since batch is open 00:00:00
	iCurrentPhaseNo						:INT;	  	//Current phase number 1/2/3....20
	iTotalPhaseNo						:INT;	  	//Total phase number 1/2/3...20
	iCurrentPhaseType					:INT;	  	//Current Phaes Type Production: 0-Feeding,1-Mixing,2-Discharge - Same for Cleaning
	sStepTime							:STRING;  	//Time elapsed in current MAIN step 00:00:00
	rStepTime1							:REAL;    	//Time elapsed in current SUB step - filling bar value
	rStepTime2							:REAL;		//Time elapsed in current SUB step - filling bar value
	rStepTime3							:REAL;		//Time elapsed in current SUB step - filling bar value
	rStepTime4							:REAL;		//Time elapsed in current SUB step - filling bar value
	rStepTime5							:REAL;		//Time elapsed in current SUB step - filling bar value
	rStepTime6							:REAL;		//Time elapsed in current SUB step - filling bar value
	rStepTime7							:REAL;		//Time elapsed in current SUB step - filling bar value
	sStepTime1							:STRING;    	//Time elapsed 00:00:00 format
	sStepTime2							:STRING;		//Time elapsed 00:00:00 format
	sStepTime3							:STRING;		//Time elapsed 00:00:00 format
	sStepTime4							:STRING;		//Time elapsed 00:00:00 format
	sStepTime5							:STRING;		//Time elapsed 00:00:00 format
	sStepTime6							:STRING;		//Time elapsed 00:00:00 format
	sStepTime7							:STRING;		//Time elapsed 00:00:00 format
	rStepTime1Prod						:REAL;
	sStepTime1Prod						:STRING;
	bBatchConfirmed1					:BOOL;		//Response from Confirmation 1 - On batch startup
	bBatchConfirmed2					:BOOL;		//Response from Confirmation 1 - On batch startup
	bBatchConfirmed3					:BOOL;		//Response from Confirmation 1 - On batch startup - NO IN PRODUCTION
	bBatchConfirmed4					:BOOL;		//Response from Confirmation 1 - On batch startup - NO IN PRODUCTION
	iFlapState							:INT; 		//0-Closed, 1-Opened, 2- Traveling, 3-Fault
	bDoorLocked							:BOOL;
	bDetergentReq						:BOOL;
	bDischargeOpenReq					:BOOL;
	bDischargeCloseReq					:BOOL;
	bBarrelInPos						:BOOL;
END_STRUCT
END_TYPE

// ---- DUTs/ST_TONP.TcDUT
TYPE ST_TONP :
STRUCT
	ET				:TIME;
	Q				:BOOL;
END_STRUCT
END_TYPE

// ---- DUTs/ST_TX_Python.TcDUT
TYPE ST_TX_Python :
STRUCT
	sAuditExportQuery				:STRING[300];
	sAuditFileName					:STRING[300];
	sBatchName						:STRING[300];
END_STRUCT
END_TYPE

// ---- Mapping/ST_EL1819.TcDUT
TYPE ST_EL1819 :
STRUCT
	Ch1_Value						AT %I*	:BOOL;
	Ch2_Value						AT %I*	:BOOL;
	Ch3_Value						AT %I*	:BOOL;
	Ch4_Value						AT %I*	:BOOL;
	Ch5_Value						AT %I*	:BOOL;
	Ch6_Value						AT %I*	:BOOL;
	Ch7_Value						AT %I*	:BOOL;
	Ch8_Value						AT %I*	:BOOL;
	Ch9_Value						AT %I*	:BOOL;
	Ch10_Value						AT %I*	:BOOL;
	Ch11_Value						AT %I*	:BOOL;
	Ch12_Value						AT %I*	:BOOL;
	Ch13_Value						AT %I*	:BOOL;
	Ch14_Value						AT %I*	:BOOL;
	Ch15_Value						AT %I*	:BOOL;
	Ch16_Value						AT %I*	:BOOL;
	State							AT %I*	:UINT;
END_STRUCT
END_TYPE

// ---- Mapping/ST_EL2809.TcDUT
TYPE ST_EL2809 :
STRUCT
	Ch1_Value						AT %Q*	:BOOL;
	Ch2_Value						AT %Q*	:BOOL;
	Ch3_Value						AT %Q*	:BOOL;
	Ch4_Value						AT %Q*	:BOOL;
	Ch5_Value						AT %Q*	:BOOL;
	Ch6_Value						AT %Q*	:BOOL;
	Ch7_Value						AT %Q*	:BOOL;
	Ch8_Value						AT %Q*	:BOOL;
	Ch9_Value						AT %Q*	:BOOL;
	Ch10_Value						AT %Q*	:BOOL;
	Ch11_Value						AT %Q*	:BOOL;
	Ch12_Value						AT %Q*	:BOOL;
	Ch13_Value						AT %Q*	:BOOL;
	Ch14_Value						AT %Q*	:BOOL;
	Ch15_Value						AT %Q*	:BOOL;
	Ch16_Value						AT %Q*	:BOOL;
	State							AT %I*	:UINT;
END_STRUCT
END_TYPE

// ---- Mapping/ST_EL3174.TcDUT
TYPE ST_EL3174 :
STRUCT
	Ch1_Error						AT %I*	:BOOL;
	Ch1_Value						AT %I*	:INT;
	Ch2_Error						AT %I*	:BOOL;
	Ch2_Value						AT %I*	:INT;
	Ch3_Error						AT %I*	:BOOL;
	Ch3_Value						AT %I*	:INT;
	Ch4_Error						AT %I*	:BOOL;
	Ch4_Value						AT %I*	:INT;
	State							AT %I*	:UINT;
END_STRUCT
END_TYPE

// ---- Mapping/ST_EL3214.TcDUT
TYPE ST_EL3214 :
STRUCT
	Ch1_Error						AT %I*	:BOOL;
	Ch1_Value						AT %I*	:INT;
	Ch2_Error						AT %I*	:BOOL;
	Ch2_Value						AT %I*	:INT;
	Ch3_Error						AT %I*	:BOOL;
	Ch3_Value						AT %I*	:INT;
	Ch4_Error						AT %I*	:BOOL;
	Ch4_Value						AT %I*	:INT;
	State							AT %I*	:UINT;
END_STRUCT
END_TYPE

// ---- Mapping/ST_EL4008.TcDUT
TYPE ST_EL4008 :
STRUCT
	Ch1_Value						AT %Q*	:INT;
	Ch2_Value						AT %Q*	:INT;
	Ch3_Value						AT %Q*	:INT;
	Ch4_Value						AT %Q*	:INT;
	Ch5_Value						AT %Q*	:INT;
	Ch6_Value						AT %Q*	:INT;
	Ch7_Value						AT %Q*	:INT;
	Ch8_Value						AT %Q*	:INT;
	State							AT %I*	:UINT;
END_STRUCT
END_TYPE

// ---- Mapping/ST_EL4124.TcDUT
TYPE ST_EL4124 :
STRUCT
	Ch1_Value						AT %Q*	:INT;
	Ch2_Value						AT %Q*	:INT;
	Ch3_Value						AT %Q*	:INT;
	Ch4_Value						AT %Q*	:INT;
	State							AT %I*	:UINT;
END_STRUCT
END_TYPE

// ---- Mapping/ST_EL6021.TcDUT
TYPE ST_EL6021 :
STRUCT
	State							AT %I*	:UINT;
END_STRUCT
END_TYPE

// ---- Mapping/ST_EL9110.TcDUT
TYPE ST_EL9110 :
STRUCT
	PowerOK							AT %I*	:BOOL;
	State							AT %I*	:UINT;
END_STRUCT
END_TYPE

// ---- GVLs/CONST.TcGVL
{attribute 'qualified_only'}
VAR_GLOBAL
	AMS_NETID					:STRING:='169.254.227.12.1.1';
	PROJECT_DIR					:STRING:='C:\TwinCAT\243702-Lodige AK\';
	DB_ID						:UDINT:=1;
END_VAR
VAR_GLOBAL PERSISTENT
	Production_Active: ST_Recipe_Production;
END_VAR

// ---- GVLs/GV.TcGVL
{attribute 'qualified_only'}
VAR_GLOBAL
	
	{attribute 'OPC.UA.DA' := '1'}
	{attribute 'OPC.UA.DA.StructuredType' := '1'}
	stOPC							:ST_OPC;	

	bIO_Card_Failure				:BOOL;

	shunt							:BOOL;
	bLogOut							:BOOL;

	sEmptyString					:STRING:='';
	
	sAdminsitratorUser				:STRING:='__SystemAdministrator';
	sDefaultUser					:STRING:='DefaultUser';
	sSystemUser						:STRING:='__SystemUser';

	stTime							:ST_Time;
	stIPCDiag						:ST_Diagnostic;	
	stHMI							:ST_HMI;
	stToHMI							:ST_ToHMI;
	

	stAlarm							:ST_Alarm;
	stReport						:ST_Report;
	
	
	stCleaningCmd					:ST_ProcessCmd;
	stProductionCmd					:ST_ProcessCmd;
	stBlowingCmd					:ST_PRocessCmd;
	stAutoProcessCmd				:ST_ProcessCmd;
	
	bFlapCloseAfterBatch			:BOOL;
	
	stTX_Python						:ST_TX_Python;
	stRX_Python						:ST_RX_Python;
	
	bMixerL_Flow_OK					:BOOL;
	bMixerR_Flow_OK					:BOOL;
	bChopper1_Flow_OK				:BOOL;
	bChopper2_Flow_OK				:BOOL;
	
	
	bAlarmOK						:BOOL;
	bMixerStopped					:BOOL;
	bDisCloseReq					:BOOL;
	bDisOpenReq						:BOOL;
	
	bUserLogged						:BOOL;
	
	iPP								:INT;
	iCP								:INT;
	
	iPrevPP							:INT;
	iPrevCP							:INT;
	
	bDisableNext					:BOOL;
	bDisablePrev					:BOOL;
	
	sProdPhases						:ARRAY[0..2] OF STRING := ['Feeding','Mixing','Discharging'];
	sCleanPhases					:ARRAY[0..6] OF STRING := ['Rinsing','Mount/Dismount','Main Clean','PW Clean','Draining','Blowing','Clean Control'];
	sChopperModes					:ARRAY[0..2] OF STRING := ['OFF','ON','ON'];
	sMixerModes						:ARRAY[0..4] OF STRING := ['OFF','ON/Forward','Interval','Backward','Alternate'];
	sEndPoints						:ARRAY[0..1] OF STRING := ['Auto','Manual'];
	sMediums						:ARRAY[0..2] OF STRING := ['Cold Water','Warm Water','Purified Water'];
	sDetergent						:ARRAY[0..2] OF STRING := ['OFF','ON','ON'];

	
	
	rMixerSpeed_AV					:REAL;
	rMixerCurrent_AV				:REAL;
	rChopper1Current_AV				:REAL;
	rChopper2Current_AV				:REAL;
	rProductTemperature_AV			:REAL;
	rProductTemperature_RAW			:REAL;
	
	rMixerLFlow_AV					:REAL;
	rMixerRFlow_AV					:REAL;
	rChopper1Flow_AV				:REAL;
	rChopper2Flow_AV				:REAL;
	


	
END_VAR
VAR_GLOBAL PERSISTENT
	stSettings						:ST_Settings;
	stBatch							:ST_Batch;
	stBatches 						:ARRAY[0..9] OF ST_Batch;
	stLastBatch						:ST_Batch;
	stControl						:ST_Control;
	sUserLogged						:STRING;
	sGroupLogged					:STRING;
	bBatchOpen						:BOOL;
	bBatchClose						:BOOL;
	bBatchBusy						:BOOL;
	iRecipeType						:INT;
END_VAR

// ---- GVLs/IN.TcGVL
{attribute 'qualified_only'}
VAR_GLOBAL
	

	bVoltageDC_Fault						:BOOL;
	bCabinetFan_Fault						:BOOL;
	bEmergencyStop							:BOOL;
	bCompressedAirOK						:BOOL;
	bDoorClosed								:BOOL;
	bDoorLocked							    :BOOL;
	
	
	bMixerFreqConv_Fault					:BOOL;
	bChopper1Protection_Fault				:BOOL;
	bChopper2Protection_Fault				:BOOL;

	bDischargeFlap_Fixed					:BOOL;
	bDischargeFlap_Opened					:BOOL;
	bDischargeFlap_Closed					:BOOL;
	bDischargeFlap_HalfOpen					:BOOL;

	
	iMixerSpeed								:INT;    //0..20mA
	iMixerCurrent							:INT; 	//0..20mA	
	iChopper1Current						:INT; 	//4..20mA
	iChopper2Current						:INT; 	//4..20mA
	iProductTemperature						:INT; 	//0..20mA 0-150 C
	
	iFlowMixerL								:INT;
	iFlowMixerR							    :INT;
	iFlowChopper1							:INT;
	iFlowChopper2							:INT;

END_VAR

// ---- GVLs/OUT.TcGVL
{attribute 'qualified_only'}
VAR_GLOBAL
	
	bDoor_Unlock					:BOOL;
	bVoltageON_Light				:BOOL;
	bMixerForward					:BOOL;
	bMixerBackward				 	:BOOL;
	bHeater						 	:BOOL;
	bChopper1					 	:BOOL;
	bChopper2					 	:BOOL;
	bDischarge_Open					:BOOL;
	bDischarge_Close		 		:BOOL;
	bDischarge_Fix					:BOOL;
	
	bDryingPipeSocket_V1010			:BOOL;
	bCleaningAir_V1030			 	:BOOL;
	bCleaningWater_V1020		 	:BOOL;
	bColdWater					 	:BOOL;
	bWarmWater					 	:BOOL;
	bTightAir_V1100					:BOOL;
	bProcessWater_V1025			 	:BOOL;
	
	bChopper1_Air_V1080		 		:BOOL;
	bChopper1_Water_V1570		 	:BOOL;
	bChopper1_Drain_V1150		 	:BOOL;
	
	bChopper2_Air_V1090		 		:BOOL;
	bChopper2_Water_V1580		 	:BOOL;
	bChopper2_Drain_V1160		 	:BOOL;
	
	bAlarm							:BOOL;
	bDoorOpen_Light				 	:BOOL;
	
	
	iMixerSpeed					 	:INT;
	
END_VAR

// ---- GVLs/Recipes.TcGVL
{attribute 'qualified_only'}
VAR_GLOBAL
	Production						:ST_Recipe_Production;
	Cleaning						:ST_Recipe_Cleaning;

	Production_Empty				:ST_Recipe_Production;
	Cleaning_Empty					:ST_Recipe_Cleaning;
	
	Production_Phase_Empty			:ST_Production_Phases;
	Cleaning_Phase_Empty			:ST_Cleaning_Phases;
	
	Production_Phase_HMI			:ST_Production_Phases;
	Cleaning_Phase_HMI				:ST_Cleaning_Phases;
	
END_VAR
VAR_GLOBAL PERSISTENT
	Production_Active				:ST_Recipe_Production;
	Cleaning_Active					:ST_Recipe_Cleaning;
END_VAR

// ---- POUs/MAIN.TcPOU
PROGRAM MAIN
VAR
	bFirstCycle				:BOOL:=TRUE;
	tonFirstCycleDelay		:TON;
	bFirstCycleDelay		:BOOL;
	
	//UPS
	fbUPS					:FB_S_UPS_BAPI;
	eGlobalSUpsState 		:E_S_UPS_State;
	fbWritePersistent		:WritePersistentData;
	
	bPowerFailure			:BOOL;
	
	//IPC diagnostic
	//fbReg					:FB_IPCDiag_Register;
	//fbIPC_Temp				:FB_IPCDiag_ReadParameter;
	//fbIPC_BootCnt			:FB_IPCDiag_ReadParameter;
	//fbIPC_OperTime			:FB_IPCDiag_ReadParameter;	
	
	//Close application	
	fbCloseHMI				:NT_StartProcess;
	fbCloseRDP				:NT_StartProcess;
	
	
	//Auto logout
	tonUserTimeOut			:TON;
	tonUserLogOut			:TON;

	sLogoutShift1			:STRING;
	sLogoutShift2			:STRING;
	sLogoutShift3			:STRING;
	
	bLogout					:BOOL;
	tonLogout				:TON;
	
	
	opcTrigMixStart			:R_TRIG;
	opcTrigMixStop			:F_TRIG;
END_VAR

P00_Mapping();
P01_AnalogScaling();
P02_GlobalSystemTime();


P1_00_MAIN();
P2_00_MAIN();
P3_00_MAIN();
P4_00_MAIN();
P5_00_MAIN();

bFirstCycle:=FALSE;

END_PROGRAM

// ---- POUs/P00_Mapping.TcPOU
PROGRAM P00_Mapping
VAR
	AI_SPARE								:INT;
	DI_SPARE								:BOOL;
	AO_SPARE								:INT:=0;
	DO_SPARE								:BOOL:=FALSE;
	
	
	TI1										:ST_EL3214;
	AI1										:ST_EL3174;
	AI2										:ST_EL3174;
	DI1										:ST_EL1819;
	AO1										:ST_EL4124;
	PS1										:ST_EL9110;
	DO1										:ST_EL2809;
	DO2										:ST_EL2809;
	PB1										:ST_EL6021;


END_VAR

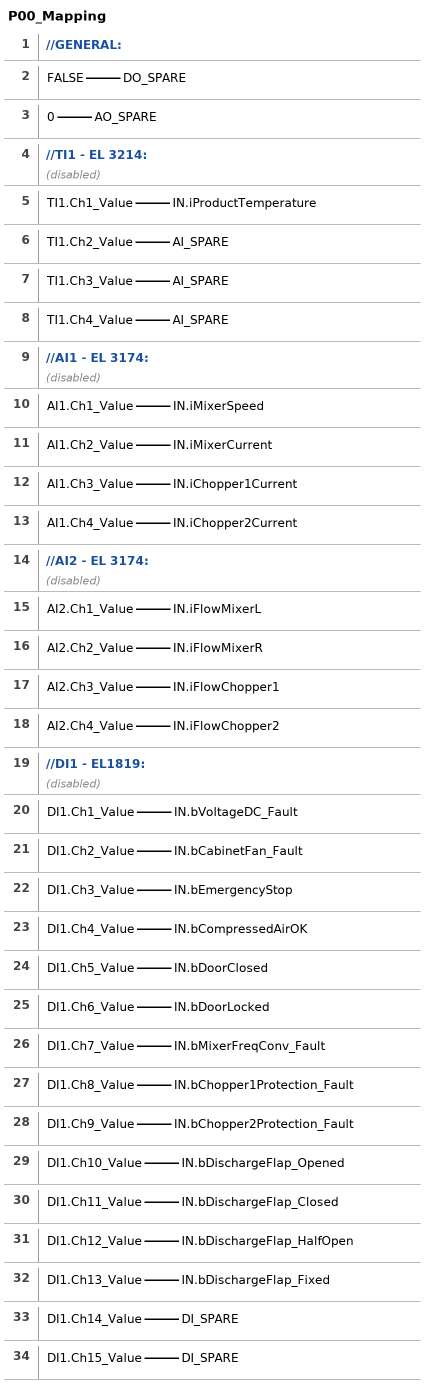
// NETWORK 1
// label: //GENERAL

// NETWORK 2
DO_SPARE := FALSE;

// NETWORK 3
AO_SPARE := 0;

// NETWORK 4 (disabled)
// label: //TI1 - EL 3214

// NETWORK 5
IN.iProductTemperature := TI1.Ch1_Value;

// NETWORK 6
AI_SPARE := TI1.Ch2_Value;

// NETWORK 7
AI_SPARE := TI1.Ch3_Value;

// NETWORK 8
AI_SPARE := TI1.Ch4_Value;

// NETWORK 9 (disabled)
// label: //AI1 - EL 3174

// NETWORK 10
IN.iMixerSpeed := AI1.Ch1_Value;

// NETWORK 11
IN.iMixerCurrent := AI1.Ch2_Value;

// NETWORK 12
IN.iChopper1Current := AI1.Ch3_Value;

// NETWORK 13
IN.iChopper2Current := AI1.Ch4_Value;

// NETWORK 14 (disabled)
// label: //AI2 - EL 3174

// NETWORK 15
IN.iFlowMixerL := AI2.Ch1_Value;

// NETWORK 16
IN.iFlowMixerR := AI2.Ch2_Value;

// NETWORK 17
IN.iFlowChopper1 := AI2.Ch3_Value;

// NETWORK 18
IN.iFlowChopper2 := AI2.Ch4_Value;

// NETWORK 19 (disabled)
// label: //DI1 - EL1819

// NETWORK 20
IN.bVoltageDC_Fault := DI1.Ch1_Value;

// NETWORK 21
IN.bCabinetFan_Fault := DI1.Ch2_Value;

// NETWORK 22
IN.bEmergencyStop := DI1.Ch3_Value;

// NETWORK 23
IN.bCompressedAirOK := DI1.Ch4_Value;

// NETWORK 24
IN.bDoorClosed := DI1.Ch5_Value;

// NETWORK 25
IN.bDoorLocked := DI1.Ch6_Value;

// NETWORK 26
IN.bMixerFreqConv_Fault := DI1.Ch7_Value;

// NETWORK 27
IN.bChopper1Protection_Fault := DI1.Ch8_Value;

// NETWORK 28
IN.bChopper2Protection_Fault := DI1.Ch9_Value;

// NETWORK 29
IN.bDischargeFlap_Opened := DI1.Ch10_Value;

// NETWORK 30
IN.bDischargeFlap_Closed := DI1.Ch11_Value;

// NETWORK 31
IN.bDischargeFlap_HalfOpen := DI1.Ch12_Value;

// NETWORK 32
IN.bDischargeFlap_Fixed := DI1.Ch13_Value;

// NETWORK 33
DI_SPARE := DI1.Ch14_Value;

// NETWORK 34
DI_SPARE := DI1.Ch15_Value;

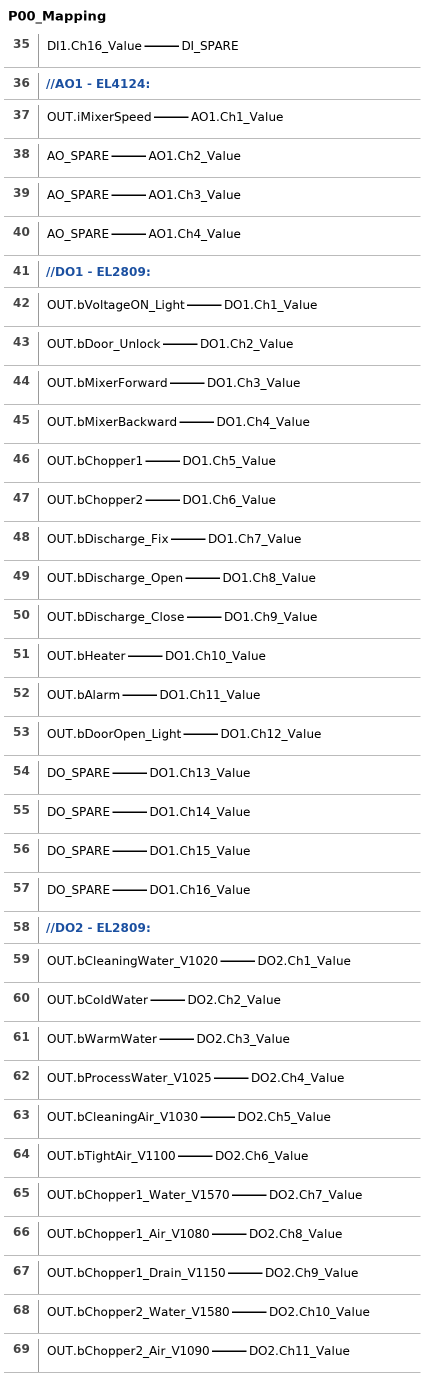
// NETWORK 35
DI_SPARE := DI1.Ch16_Value;

// NETWORK 36
// label: //AO1 - EL4124

// NETWORK 37
AO1.Ch1_Value := OUT.iMixerSpeed;

// NETWORK 38
AO1.Ch2_Value := AO_SPARE;

// NETWORK 39
AO1.Ch3_Value := AO_SPARE;

// NETWORK 40
AO1.Ch4_Value := AO_SPARE;

// NETWORK 41
// label: //DO1 - EL2809

// NETWORK 42
DO1.Ch1_Value := OUT.bVoltageON_Light;

// NETWORK 43
DO1.Ch2_Value := OUT.bDoor_Unlock;

// NETWORK 44
DO1.Ch3_Value := OUT.bMixerForward;

// NETWORK 45
DO1.Ch4_Value := OUT.bMixerBackward;

// NETWORK 46
DO1.Ch5_Value := OUT.bChopper1;

// NETWORK 47
DO1.Ch6_Value := OUT.bChopper2;

// NETWORK 48
DO1.Ch7_Value := OUT.bDischarge_Fix;

// NETWORK 49
DO1.Ch8_Value := OUT.bDischarge_Open;

// NETWORK 50
DO1.Ch9_Value := OUT.bDischarge_Close;

// NETWORK 51
DO1.Ch10_Value := OUT.bHeater;

// NETWORK 52
DO1.Ch11_Value := OUT.bAlarm;

// NETWORK 53
DO1.Ch12_Value := OUT.bDoorOpen_Light;

// NETWORK 54
DO1.Ch13_Value := DO_SPARE;

// NETWORK 55
DO1.Ch14_Value := DO_SPARE;

// NETWORK 56
DO1.Ch15_Value := DO_SPARE;

// NETWORK 57
DO1.Ch16_Value := DO_SPARE;

// NETWORK 58
// label: //DO2 - EL2809

// NETWORK 59
DO2.Ch1_Value := OUT.bCleaningWater_V1020;

// NETWORK 60
DO2.Ch2_Value := OUT.bColdWater;

// NETWORK 61
DO2.Ch3_Value := OUT.bWarmWater;

// NETWORK 62
DO2.Ch4_Value := OUT.bProcessWater_V1025;

// NETWORK 63
DO2.Ch5_Value := OUT.bCleaningAir_V1030;

// NETWORK 64
DO2.Ch6_Value := OUT.bTightAir_V1100;

// NETWORK 65
DO2.Ch7_Value := OUT.bChopper1_Water_V1570;

// NETWORK 66
DO2.Ch8_Value := OUT.bChopper1_Air_V1080;

// NETWORK 67
DO2.Ch9_Value := OUT.bChopper1_Drain_V1150;

// NETWORK 68
DO2.Ch10_Value := OUT.bChopper2_Water_V1580;

// NETWORK 69
DO2.Ch11_Value := OUT.bChopper2_Air_V1090;

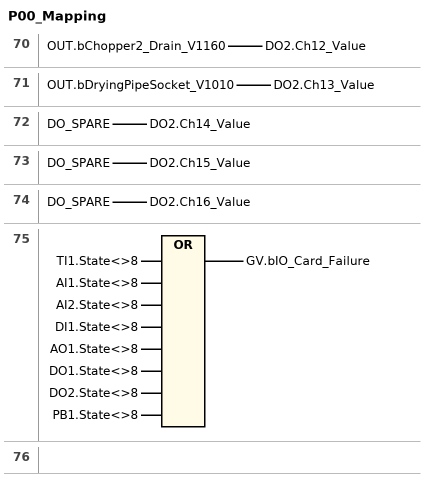
// NETWORK 70
DO2.Ch12_Value := OUT.bChopper2_Drain_V1160;

// NETWORK 71
DO2.Ch13_Value := OUT.bDryingPipeSocket_V1010;

// NETWORK 72
DO2.Ch14_Value := DO_SPARE;

// NETWORK 73
DO2.Ch15_Value := DO_SPARE;

// NETWORK 74
DO2.Ch16_Value := DO_SPARE;

// NETWORK 75
GV.bIO_Card_Failure := (TI1.State<>8) OR (AI1.State<>8) OR (AI2.State<>8) OR (DI1.State<>8) OR (AO1.State<>8) OR (DO1.State<>8) OR (DO2.State<>8) OR (PB1.State<>8);

// NETWORK 76

END_PROGRAM

// ---- POUs/P01_AnalogScaling.TcPOU
PROGRAM P01_AnalogScaling
VAR
	fbMixerSpeed				:FB_Scale;
	fbMixerSpeed2				:FB_Scale;
	fbMixerSpeed_AVG			:FB_AVG200;
	fbMixerCurrent				:FB_Scale;
	fbMixerCurrent_AVG			:FB_AVG200;
	
	fbChopper1Current			:FB_Scale;
	fbChopper1Current_AVG		:FB_AVG200;
	fbChopper2Current			:FB_Scale;
	fbChopper2Current_AVG		:FB_AVG200;
	
	fbProductTemperature		:FB_Scale;
	fbProductTemperature_AVG	:FB_AVG200;
	
	fbFlowMixerL				:FB_Scale;
	fbFlowMixerR				:FB_Scale;
	fbFlowChopper1				:FB_Scale;
	fbFlowChopper2				:FB_Scale;
	
	fbFlowMixerL_AVG			:FB_AVG200;
	fbFlowMixerR_AVG			:FB_AVG200;
	fbFlowChopper1_AVG			:FB_AVG200;
	fbFlowChopper2_AVG			:FB_AVG200;
	
	rOffset1					:REAL;
	fbChopper2Current2: FB_Scale;
	
	TON_SpeedRamp				:TON;
	tofMixerAV: TOF;
END_VAR

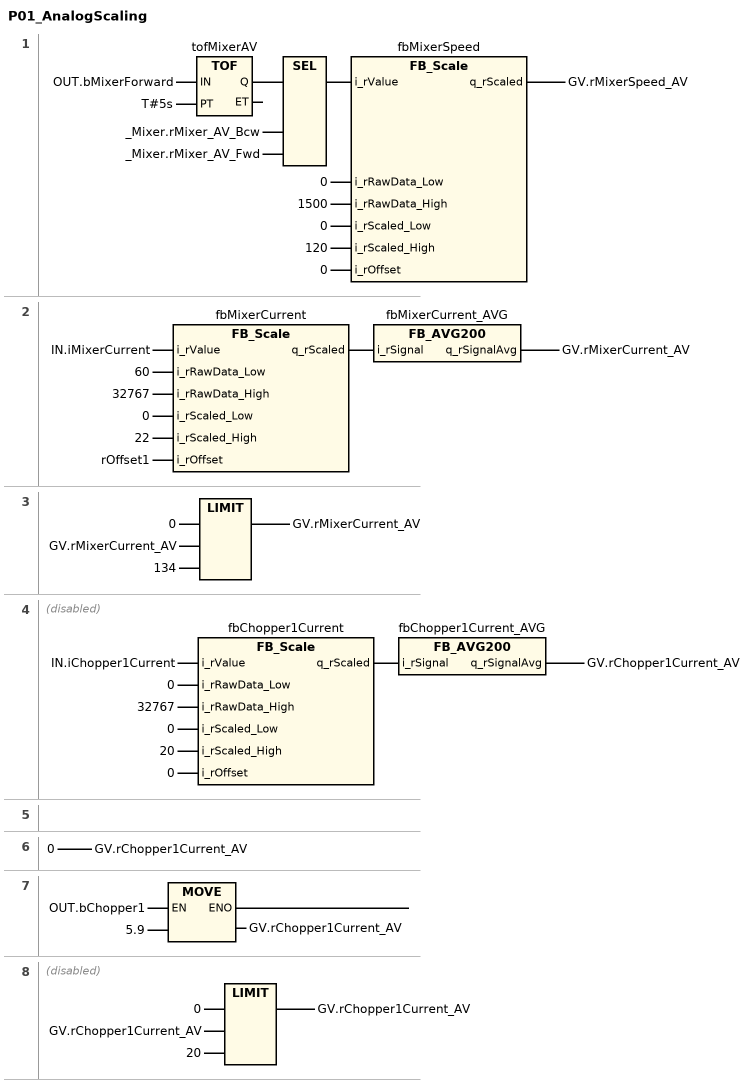
// NETWORK 1
tofMixerAV(IN := OUT.bMixerForward, PT := T#5s); // TOF
fbMixerSpeed(
    i_rValue := SEL(tofMixerAV.Q, _Mixer.rMixer_AV_Bcw, _Mixer.rMixer_AV_Fwd),
    i_rRawData_Low := 0,
    i_rRawData_High := 1500,
    i_rScaled_Low := 0,
    i_rScaled_High := 120,
    i_rOffset := 0); // FB_Scale
GV.rMixerSpeed_AV := fbMixerSpeed.q_rScaled;

// NETWORK 2
fbMixerCurrent(
    i_rValue := IN.iMixerCurrent,
    i_rRawData_Low := 60,
    i_rRawData_High := 32767,
    i_rScaled_Low := 0,
    i_rScaled_High := 22,
    i_rOffset := rOffset1); // FB_Scale
fbMixerCurrent_AVG(i_rSignal := fbMixerCurrent.q_rScaled); // FB_AVG200
GV.rMixerCurrent_AV := fbMixerCurrent_AVG.q_rSignalAvg;

// NETWORK 3
GV.rMixerCurrent_AV := LIMIT(0, GV.rMixerCurrent_AV, 134);

// NETWORK 4 (disabled)
// fbChopper1Current(
//     i_rValue := IN.iChopper1Current,
//     i_rRawData_Low := 0,
//     i_rRawData_High := 32767,
//     i_rScaled_Low := 0,
//     i_rScaled_High := 20,
//     i_rOffset := 0); // FB_Scale
// fbChopper1Current_AVG(i_rSignal := fbChopper1Current.q_rScaled); // FB_AVG200
// GV.rChopper1Current_AV := fbChopper1Current_AVG.q_rSignalAvg;

// NETWORK 5

// NETWORK 6
GV.rChopper1Current_AV := 0;

// NETWORK 7
IF OUT.bChopper1 THEN GV.rChopper1Current_AV := 5.9; END_IF

// NETWORK 8 (disabled)
// GV.rChopper1Current_AV := LIMIT(0, GV.rChopper1Current_AV, 20);

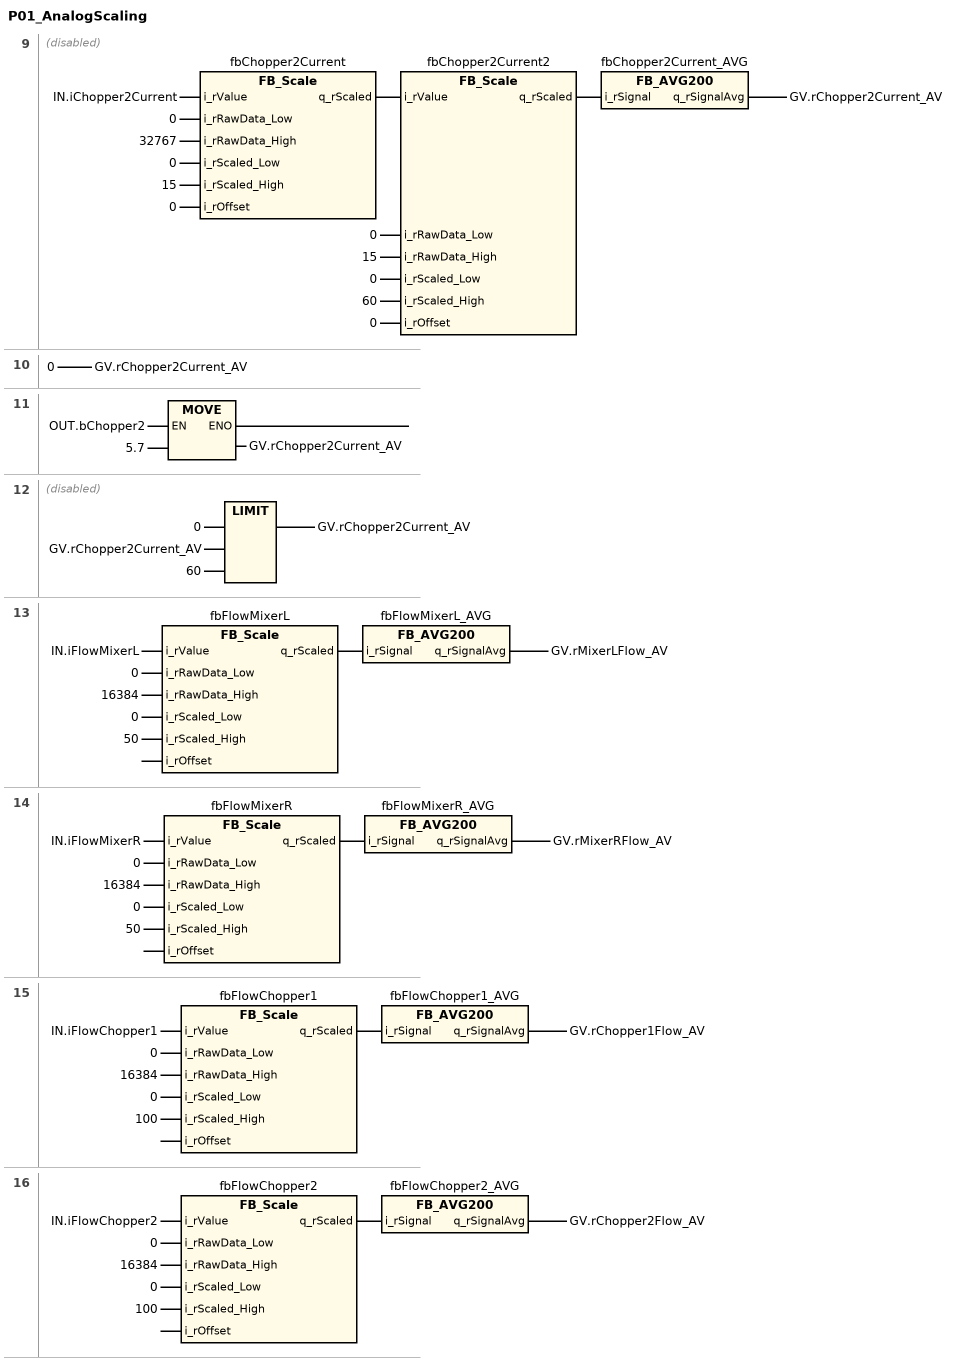
// NETWORK 9 (disabled)
// fbChopper2Current(
//     i_rValue := IN.iChopper2Current,
//     i_rRawData_Low := 0,
//     i_rRawData_High := 32767,
//     i_rScaled_Low := 0,
//     i_rScaled_High := 15,
//     i_rOffset := 0); // FB_Scale
// fbChopper2Current2(
//     i_rValue := fbChopper2Current.q_rScaled,
//     i_rRawData_Low := 0,
//     i_rRawData_High := 15,
//     i_rScaled_Low := 0,
//     i_rScaled_High := 60,
//     i_rOffset := 0); // FB_Scale
// fbChopper2Current_AVG(i_rSignal := fbChopper2Current2.q_rScaled); // FB_AVG200
// GV.rChopper2Current_AV := fbChopper2Current_AVG.q_rSignalAvg;

// NETWORK 10
GV.rChopper2Current_AV := 0;

// NETWORK 11
IF OUT.bChopper2 THEN GV.rChopper2Current_AV := 5.7; END_IF

// NETWORK 12 (disabled)
// GV.rChopper2Current_AV := LIMIT(0, GV.rChopper2Current_AV, 60);

// NETWORK 13
fbFlowMixerL(
    i_rValue := IN.iFlowMixerL,
    i_rRawData_Low := 0,
    i_rRawData_High := 16384,
    i_rScaled_Low := 0,
    i_rScaled_High := 50); // FB_Scale
fbFlowMixerL_AVG(i_rSignal := fbFlowMixerL.q_rScaled); // FB_AVG200
GV.rMixerLFlow_AV := fbFlowMixerL_AVG.q_rSignalAvg;

// NETWORK 14
fbFlowMixerR(
    i_rValue := IN.iFlowMixerR,
    i_rRawData_Low := 0,
    i_rRawData_High := 16384,
    i_rScaled_Low := 0,
    i_rScaled_High := 50); // FB_Scale
fbFlowMixerR_AVG(i_rSignal := fbFlowMixerR.q_rScaled); // FB_AVG200
GV.rMixerRFlow_AV := fbFlowMixerR_AVG.q_rSignalAvg;

// NETWORK 15
fbFlowChopper1(
    i_rValue := IN.iFlowChopper1,
    i_rRawData_Low := 0,
    i_rRawData_High := 16384,
    i_rScaled_Low := 0,
    i_rScaled_High := 100); // FB_Scale
fbFlowChopper1_AVG(i_rSignal := fbFlowChopper1.q_rScaled); // FB_AVG200
GV.rChopper1Flow_AV := fbFlowChopper1_AVG.q_rSignalAvg;

// NETWORK 16
fbFlowChopper2(
    i_rValue := IN.iFlowChopper2,
    i_rRawData_Low := 0,
    i_rRawData_High := 16384,
    i_rScaled_Low := 0,
    i_rScaled_High := 100); // FB_Scale
fbFlowChopper2_AVG(i_rSignal := fbFlowChopper2.q_rScaled); // FB_AVG200
GV.rChopper2Flow_AV := fbFlowChopper2_AVG.q_rSignalAvg;

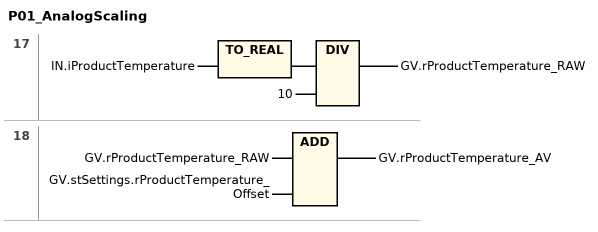
// NETWORK 17
GV.rProductTemperature_RAW := TO_REAL(IN.iProductTemperature) / 10;

// NETWORK 18
GV.rProductTemperature_AV := GV.rProductTemperature_RAW + GV.stSettings.rProductTemperature_Offset;

END_PROGRAM

// ---- FB/FB_Scale.TcPOU
// Created by Jovica Blagojeski 13.01.2022
// JB: If not known, raw data should be from 0 to 32767 (whole positive integer range), otherwise the known calibration range (highest and lowest)
// Edited by Dimitar stojanov 06.2023
// DS: Offset is added for small corrections, declaration names of variables are changed corresponding new template i_ stands for block input parameter, q_ stands for block output paramter.


//Functionality: Use this block to Scale Analog Inputs or some other Lienarization

FUNCTION_BLOCK FB_Scale
VAR_INPUT
	i_rValue 				:REAL;
	i_rRawData_Low			:REAL := 0;
	i_rRawData_High 		:REAL := 32767;
	i_rScaled_Low			:REAL:= 0;
	i_rScaled_High			:REAL:= 32767;
	i_rOffset 				:REAL;
	
END_VAR
VAR_OUTPUT
	q_rScaled 				:REAL;
END_VAR
VAR
	K 						:REAL;
	rInput 					:REAL;
END_VAR

K := ((i_rScaled_High - i_rScaled_Low) /(i_rRawData_High - i_rRawData_Low));
rInput:=i_rValue - i_rRawData_Low ;
q_rScaled:=(K * rInput) +  i_rScaled_Low + i_rOffset;

END_FUNCTION_BLOCK

// ---- FB/FB_AVG200.TcPOU
//Created by Dimitar Stojanov 06.2023

//Functionality: Calculate average value of the last 200 input samples, use for analog inputs that affectc PID regulation.

FUNCTION_BLOCK FB_AVG200
VAR_INPUT
	i_rSignal			:REAL;
END_VAR
VAR_OUTPUT
	q_rSignalAvg		:REAL;
END_VAR
VAR
	arrSignals			:ARRAY[0..199] OF REAL;
	i					:INT;
	j					:INT;
	k					:INT;
	Sum					:REAL;
END_VAR

FOR k:=0 TO 198 DO
	arrSignals[k]:=arrSignals[k+1];
END_FOR
arrSignals[199]:=i_rSignal;
Sum:=0;
FOR j:=0 TO 199 DO
	Sum := Sum + arrSignals[j];
END_FOR
IF Sum <> 0 THEN
	q_rSignalAvg:=Sum/200;
END_IF

END_FUNCTION_BLOCK

// ---- POUs/2. Process/_Mixer.TcPOU
PROGRAM _Mixer
VAR_INPUT
	i_iOperation			:INT;
	i_rSetSpeed				:REAL;
	i_rActualSpeed			:REAL;
	i_bRun					:BOOL;
	i_tIntervalFwd			:TIME;
	i_tIntervalPause		:TIME;
	i_tAlternateON			:TIME;
	i_tAlternatePause		:TIME;
END_VAR

VAR
	tonIntervalFwd			:TON;
	tonIntervalPause		:TON;
	tonAlternateON			:TON;
	tonAlternatePause		:TON;
	iStepI					:INT;
	iStepA					:INT;
	

	fbModbus				:ModbusRtuMaster_KL6x22B;
	bRead					:BOOL;
	wReadValue				:ARRAY[0..1] OF WORD;
	rMixer_AV_Fwd			:REAL;
	rMixer_AV_Bcw			:REAL;
	tonRead					:TON;
END_VAR

VAR_OUTPUT
	q_rSpeed_Cmd					:REAL;
	q_bFwd_Cmd						:BOOL;
	q_bBcw_Cmd						:BOOL;
END_VAR

IF i_iOperation = 0 THEN
	q_bBcw_Cmd:=FALSE;
	q_bFwd_Cmd:=FALSE;
ELSIF i_iOperation = 1 THEN
	q_bBcw_Cmd:=FALSE;
	q_bFwd_Cmd:=TRUE;
ELSIF i_iOperation = 2 THEN
	tonIntervalFwd(IN:=(iStepI=10),PT:=i_tIntervalFwd);
	tonIntervalPause(IN:=(iStepI=0) AND NOT i_bRun,PT:=i_tIntervalPause);
	CASE iStepI OF
		0:
			q_bBcw_Cmd:=FALSE;
			q_bFwd_Cmd:=FALSE;
			IF tonIntervalPause.Q THEN
				iStepI:=10;
			END_IF
		10:
			q_bBcw_Cmd:=FALSE;
			q_bFwd_Cmd:=TRUE;
			IF tonIntervalFwd.Q THEN
				iStepI:=0;	
			END_IF
	END_CASE
	
ELSIF i_iOperation = 3 THEN
	q_bFwd_Cmd:=FALSE;
	q_bBcw_Cmd:=TRUE;	
ELSIF i_iOperation = 4 THEN
	tonAlternateON(IN:=(iStepA=10)OR(iStepA=30),PT:=i_tAlternateON);
	tonAlternatePause(IN:=((iStepA=0)OR(iStepA=20) AND NOT i_bRun),PT:=i_tAlternatePause);
	
	CASE iStepA OF 
		0:
		   q_bBcw_Cmd:=FALSE;
		   q_bFwd_Cmd:=FALSE;
		   IF tonAlternatePause.Q THEN
			   iStepA:=10;
		   END_IF
		   
		10:
			q_bBcw_Cmd:=FALSE;
		    q_bFwd_Cmd:=TRUE;
			IF tonAlternateON.Q THEN
				iStepA:=20;
			END_IF
			
		20:
			q_bBcw_Cmd:=FALSE;
		    q_bFwd_Cmd:=FALSE;
		    IF tonAlternatePause.Q THEN
			    iStepA:=30;
		    END_IF
			
		30:
			q_bFwd_Cmd:=FALSE;
		    q_bBcw_Cmd:=TRUE;
			IF tonAlternateON.Q THEN
				iStepA:=0;
			END_IF
	END_CASE
END_IF

IF i_iOperation <> 2 THEN
	iStepI:=0;
END_IF

IF i_iOperation <> 4 THEN
	iStepA:=0;
END_IF

q_rSpeed_Cmd:=i_rSetSpeed;

MODBUS();

ACTION MODBUS:
fbModbus.ReadRegs(
				UnitID:=1,
				Quantity:= 2, 
				MBAddr:= 16169,
				cbLength:=SIZEOF(wReadValue),
				pMemoryAddr:=ADR(wReadValue),
				Execute:=bRead,
				TimeOut:=T#100MS);

bRead:=FALSE;
IF NOT fbModBus.BUSY THEN
	fbModbus.ReadRegs(Execute:=FALSE);
END_IF

tonRead(IN:=NOT(fbModBus.BUSY),PT:=T#500MS);
IF tonRead.Q THEN
	bRead:=TRUE;
END_IF

rMixer_AV_Fwd:=wReadValue[0] + wReadValue[1];

rMixer_AV_Bcw:=wReadValue[0] - wReadValue[1];
END_ACTION

END_PROGRAM

// ---- POUs/P02_GlobalSystemTime.TcPOU
PROGRAM P02_GlobalSystemTime
VAR
	fbGlobalTime 		:FB_SystemDateTIme;
END_VAR

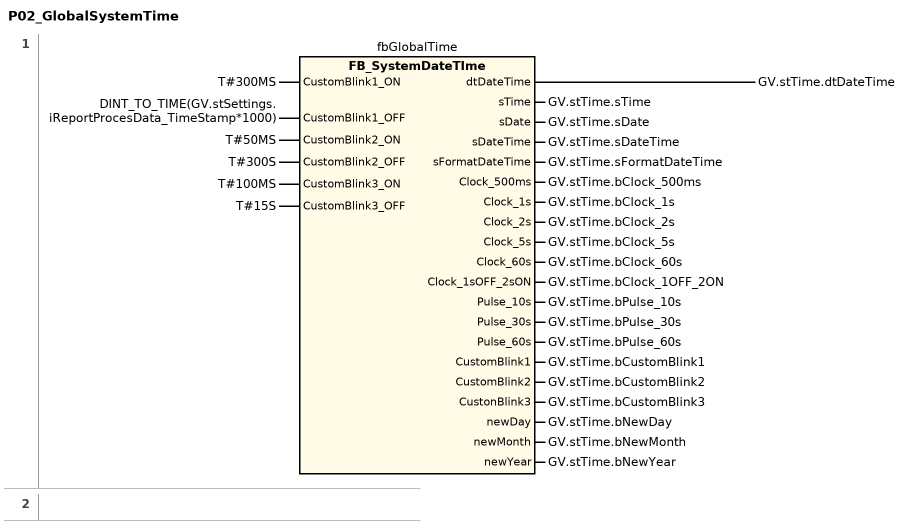
// NETWORK 1
fbGlobalTime(
    CustomBlink1_ON := T#300MS,
    CustomBlink1_OFF := DINT_TO_TIME(GV.stSettings.iReportProcesData_TimeStamp*1000),
    CustomBlink2_ON := T#50MS,
    CustomBlink2_OFF := T#300S,
    CustomBlink3_ON := T#100MS,
    CustomBlink3_OFF := T#15S,
    sTime => GV.stTime.sTime,
    sDate => GV.stTime.sDate,
    sDateTime => GV.stTime.sDateTime,
    sFormatDateTime => GV.stTime.sFormatDateTime,
    Clock_500ms => GV.stTime.bClock_500ms,
    Clock_1s => GV.stTime.bClock_1s,
    Clock_2s => GV.stTime.bClock_2s,
    Clock_5s => GV.stTime.bClock_5s,
    Clock_60s => GV.stTime.bClock_60s,
    Clock_1sOFF_2sON => GV.stTime.bClock_1OFF_2ON,
    Pulse_10s => GV.stTime.bPulse_10s,
    Pulse_30s => GV.stTime.bPulse_30s,
    Pulse_60s => GV.stTime.bPulse_60s,
    CustomBlink1 => GV.stTime.bCustomBlink1,
    CustomBlink2 => GV.stTime.bCustomBlink2,
    CustonBlink3 => GV.stTime.bCustomBlink3,
    newDay => GV.stTime.bNewDay,
    newMonth => GV.stTime.bNewMonth,
    newYear => GV.stTime.bNewYear); // FB_SystemDateTIme
GV.stTime.dtDateTime := fbGlobalTime.dtDateTime;

// NETWORK 2

END_PROGRAM

// ---- FB/FB_SystemDateTime.TcPOU
// Created by Dimitar Stojanov 06.2023 
// Install TC2_Utilities and Import ST_Time structure for fully functionality of this block


FUNCTION_BLOCK FB_SystemDateTime
VAR_INPUT
	CustomBlink1_ON		:TIME;
	CustomBlink1_OFF	:TIME;
	CustomBlink2_ON		:TIME;
	CustomBlink2_OFF	:TIME;
	CustomBlink3_ON		:TIME;
	CustomBlink3_OFF	:TIME;
END_VAR
VAR_OUTPUT
	dtDateTime		:DT;
	sTime			:STRING;
	sDate			:STRING;
	sDateTime		:STRING;
	sFormatDateTime	:STRING;
	Clock_500ms		:BOOL;
	Clock_1s		:BOOL;
	Clock_2s		:BOOL;
	Clock_5s		:BOOL;
	Clock_60s		:BOOL;
	Clock_1sOFF_2sON	:BOOL;
	Pulse_10s		:BOOL;
	Pulse_30s		:BOOL;
	Pulse_60s		:BOOL;
	CustomBlink1	:BOOL;
	CustomBlink2	:BOOL;
	CustonBlink3	:BOOL;
	newDay			:BOOL;
	newMonth		:BOOL;
	newYear			:BOOL;
END_VAR
VAR
	bFirstCycle		:BOOL:=TRUE;	

	fbTime			:FB_LocalSystemTime;
	systemDateTime	:TIMESTRUCT;
	
	Second			:STRING;
	Minute			:STRING;
	Hour			:STRING;
	Day				:STRING;
	Month			:STRING;
	Year			:STRING;
	
	iClock1s		:INT;
	TON_0: TON;
	TOF_0: TOF;
	TON_1: TON;
	TOF_1: TOF;
	TOF_2: TOF;
	TON_2: TON;
	TON_3: TON;
	TOF_3: TOF;
	TOF_4: TOF;
	TON_4: TON;
	TON_5: TON;
	TOF_5: TOF;
	TON_6: TON;
	TOF_6: TOF;
	TON_7: TON;
	TOF_7: TOF;
	TON_8: TON;
	TOF_8: TOF;
	
	TON_9: TON;
	TOF_9: TOF;
	TOF_10: TOF;
	TOF_11: TOF;
	TON_10: TON;
	TON_20: TON;
	TOF_20: TOF;
	TON_21: TON;
	TOF_21: TOF;
	TON_22: TON;
	TOF_22: TOF;
	
	bDelay			:BOOL;
	TON_DELAY		:TON;
END_VAR

VAR PERSISTENT
	CurrentDay		:WORD;
	CurrentMonth	:WORD;
	CurrentYear		:WORD;
END_VAR

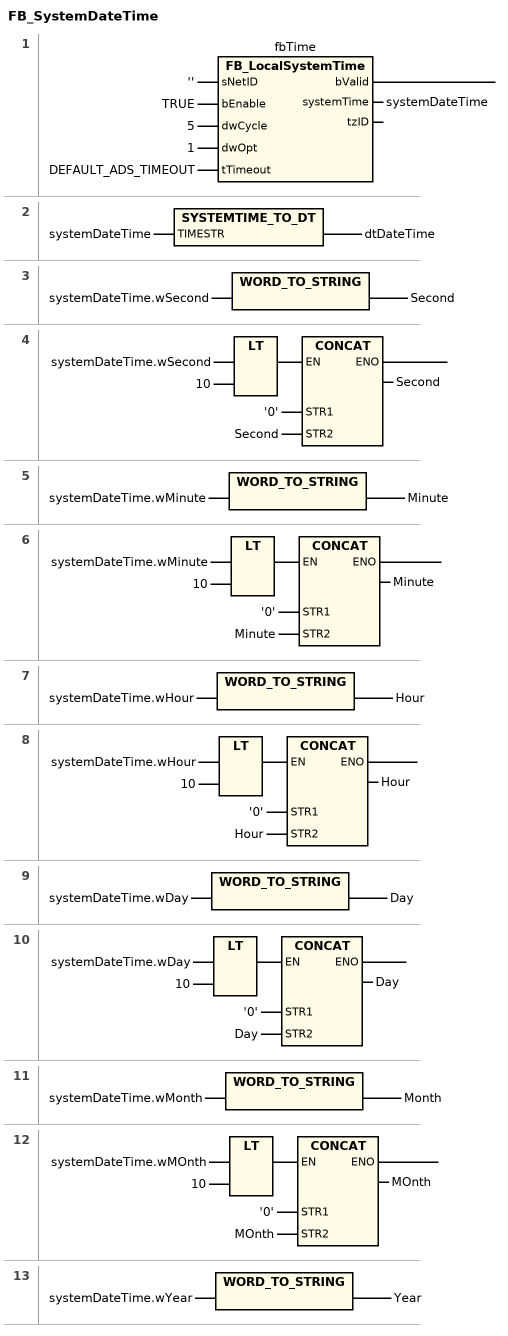
// NETWORK 1
fbTime(
    sNetID := '',
    bEnable := TRUE,
    dwCycle := 5,
    dwOpt := 1,
    tTimeout := DEFAULT_ADS_TIMEOUT,
    systemTime => systemDateTime); // FB_LocalSystemTime

// NETWORK 2
dtDateTime := SYSTEMTIME_TO_DT(TIMESTR := systemDateTime);

// NETWORK 3
Second := WORD_TO_STRING(systemDateTime.wSecond);

// NETWORK 4
IF systemDateTime.wSecond < 10 THEN Second := CONCAT(STR1 := '0', STR2 := Second); END_IF

// NETWORK 5
Minute := WORD_TO_STRING(systemDateTime.wMinute);

// NETWORK 6
IF systemDateTime.wMinute < 10 THEN Minute := CONCAT(STR1 := '0', STR2 := Minute); END_IF

// NETWORK 7
Hour := WORD_TO_STRING(systemDateTime.wHour);

// NETWORK 8
IF systemDateTime.wHour < 10 THEN Hour := CONCAT(STR1 := '0', STR2 := Hour); END_IF

// NETWORK 9
Day := WORD_TO_STRING(systemDateTime.wDay);

// NETWORK 10
IF systemDateTime.wDay < 10 THEN Day := CONCAT(STR1 := '0', STR2 := Day); END_IF

// NETWORK 11
Month := WORD_TO_STRING(systemDateTime.wMonth);

// NETWORK 12
IF systemDateTime.wMOnth < 10 THEN MOnth := CONCAT(STR1 := '0', STR2 := MOnth); END_IF

// NETWORK 13
Year := WORD_TO_STRING(systemDateTime.wYear);

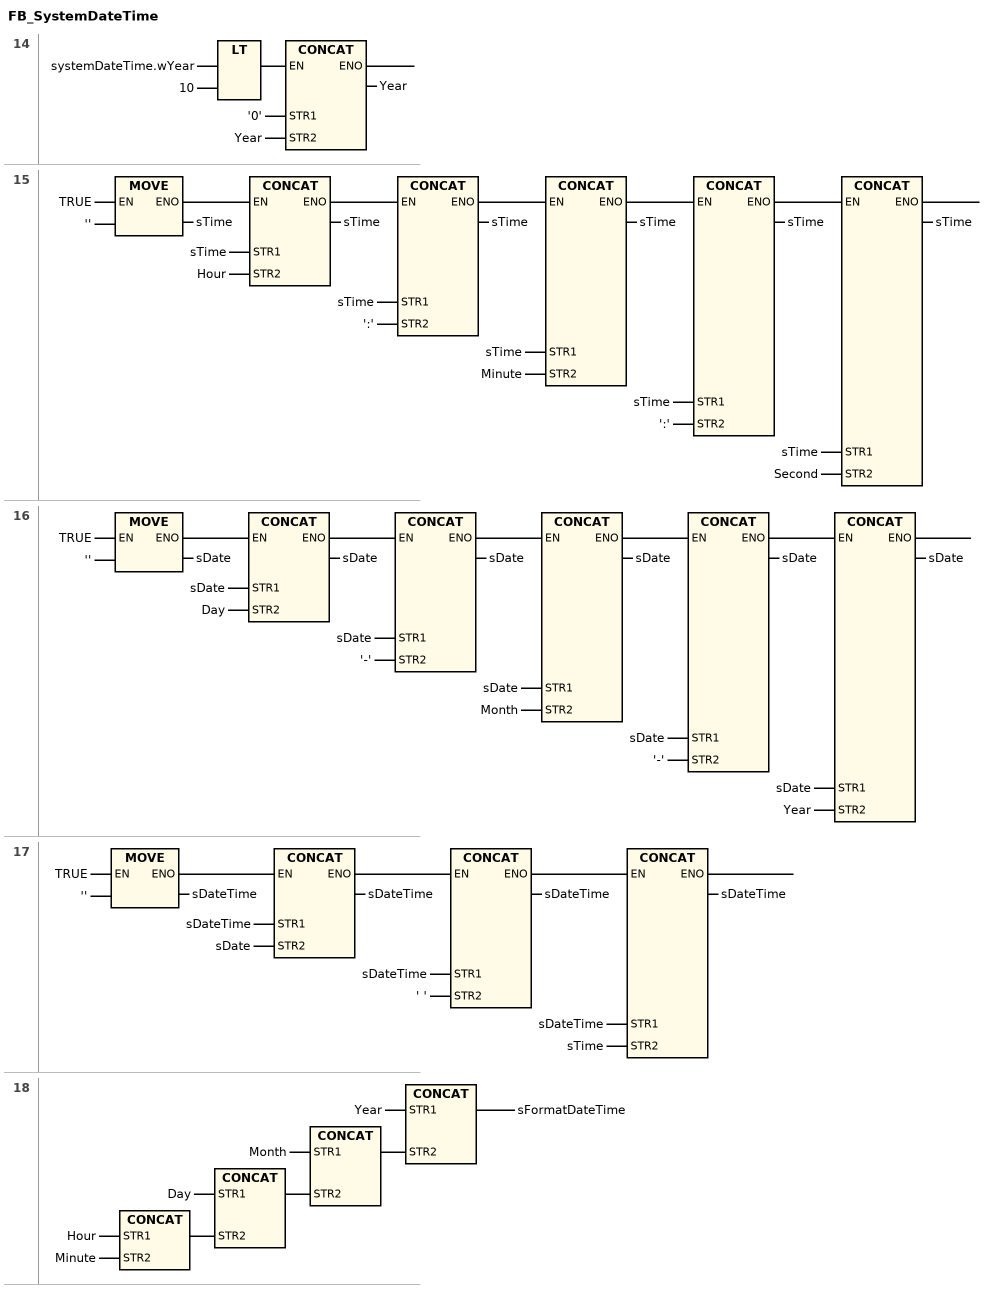
// NETWORK 14
IF systemDateTime.wYear < 10 THEN Year := CONCAT(STR1 := '0', STR2 := Year); END_IF

// NETWORK 15
sTime := '';
sTime := CONCAT(STR1 := sTime, STR2 := Hour);
sTime := CONCAT(STR1 := sTime, STR2 := ':');
sTime := CONCAT(STR1 := sTime, STR2 := Minute);
sTime := CONCAT(STR1 := sTime, STR2 := ':');
sTime := CONCAT(STR1 := sTime, STR2 := Second);

// NETWORK 16
sDate := '';
sDate := CONCAT(STR1 := sDate, STR2 := Day);
sDate := CONCAT(STR1 := sDate, STR2 := '-');
sDate := CONCAT(STR1 := sDate, STR2 := Month);
sDate := CONCAT(STR1 := sDate, STR2 := '-');
sDate := CONCAT(STR1 := sDate, STR2 := Year);

// NETWORK 17
sDateTime := '';
sDateTime := CONCAT(STR1 := sDateTime, STR2 := sDate);
sDateTime := CONCAT(STR1 := sDateTime, STR2 := ' ');
sDateTime := CONCAT(STR1 := sDateTime, STR2 := sTime);

// NETWORK 18
sFormatDateTime := CONCAT(STR1 := Year, STR2 := CONCAT(STR1 := Month, STR2 := CONCAT(STR1 := Day, STR2 := CONCAT(STR1 := Hour, STR2 := Minute))));

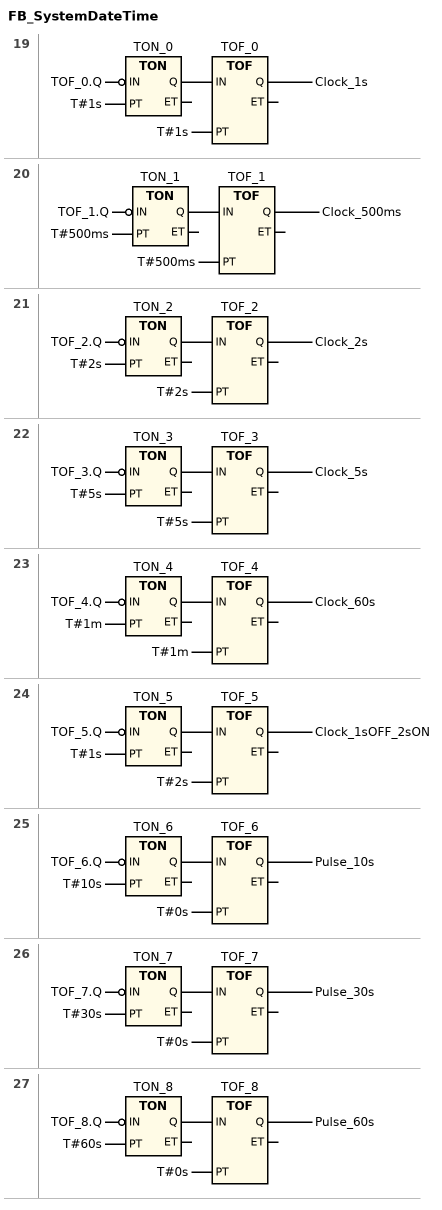
// NETWORK 19
TON_0(IN := NOT TOF_0.Q, PT := T#1s); // TON
TOF_0(IN := TON_0.Q, PT := T#1s); // TOF
Clock_1s := TOF_0.Q;

// NETWORK 20
TON_1(IN := NOT TOF_1.Q, PT := T#500ms); // TON
TOF_1(IN := TON_1.Q, PT := T#500ms); // TOF
Clock_500ms := TOF_1.Q;

// NETWORK 21
TON_2(IN := NOT TOF_2.Q, PT := T#2s); // TON
TOF_2(IN := TON_2.Q, PT := T#2s); // TOF
Clock_2s := TOF_2.Q;

// NETWORK 22
TON_3(IN := NOT TOF_3.Q, PT := T#5s); // TON
TOF_3(IN := TON_3.Q, PT := T#5s); // TOF
Clock_5s := TOF_3.Q;

// NETWORK 23
TON_4(IN := NOT TOF_4.Q, PT := T#1m); // TON
TOF_4(IN := TON_4.Q, PT := T#1m); // TOF
Clock_60s := TOF_4.Q;

// NETWORK 24
TON_5(IN := NOT TOF_5.Q, PT := T#1s); // TON
TOF_5(IN := TON_5.Q, PT := T#2s); // TOF
Clock_1sOFF_2sON := TOF_5.Q;

// NETWORK 25
TON_6(IN := NOT TOF_6.Q, PT := T#10s); // TON
TOF_6(IN := TON_6.Q, PT := T#0s); // TOF
Pulse_10s := TOF_6.Q;

// NETWORK 26
TON_7(IN := NOT TOF_7.Q, PT := T#30s); // TON
TOF_7(IN := TON_7.Q, PT := T#0s); // TOF
Pulse_30s := TOF_7.Q;

// NETWORK 27
TON_8(IN := NOT TOF_8.Q, PT := T#60s); // TON
TOF_8(IN := TON_8.Q, PT := T#0s); // TOF
Pulse_60s := TOF_8.Q;

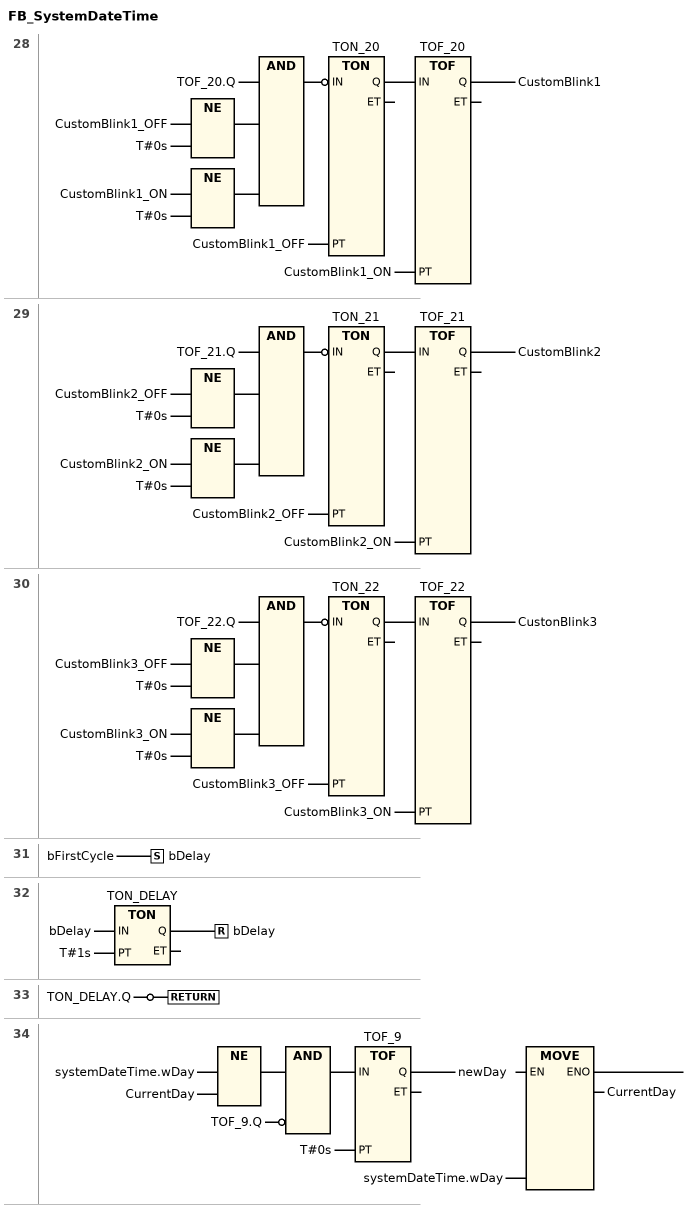
// NETWORK 28
TON_20(IN := NOT (TOF_20.Q AND CustomBlink1_OFF <> T#0s AND CustomBlink1_ON <> T#0s), PT := CustomBlink1_OFF); // TON
TOF_20(IN := TON_20.Q, PT := CustomBlink1_ON); // TOF
CustomBlink1 := TOF_20.Q;

// NETWORK 29
TON_21(IN := NOT (TOF_21.Q AND CustomBlink2_OFF <> T#0s AND CustomBlink2_ON <> T#0s), PT := CustomBlink2_OFF); // TON
TOF_21(IN := TON_21.Q, PT := CustomBlink2_ON); // TOF
CustomBlink2 := TOF_21.Q;

// NETWORK 30
TON_22(IN := NOT (TOF_22.Q AND CustomBlink3_OFF <> T#0s AND CustomBlink3_ON <> T#0s), PT := CustomBlink3_OFF); // TON
TOF_22(IN := TON_22.Q, PT := CustomBlink3_ON); // TOF
CustonBlink3 := TOF_22.Q;

// NETWORK 31
bDelay S= bFirstCycle;

// NETWORK 32
TON_DELAY(IN := bDelay, PT := T#1s); // TON
bDelay R= TON_DELAY.Q;

// NETWORK 33
IF NOT TON_DELAY.Q THEN RETURN; END_IF

// NETWORK 34
TOF_9(IN := systemDateTime.wDay <> CurrentDay AND NOT TOF_9.Q, PT := T#0s); // TOF
newDay := TOF_9.Q;
IF TOF_9.Q THEN CurrentDay := systemDateTime.wDay; END_IF

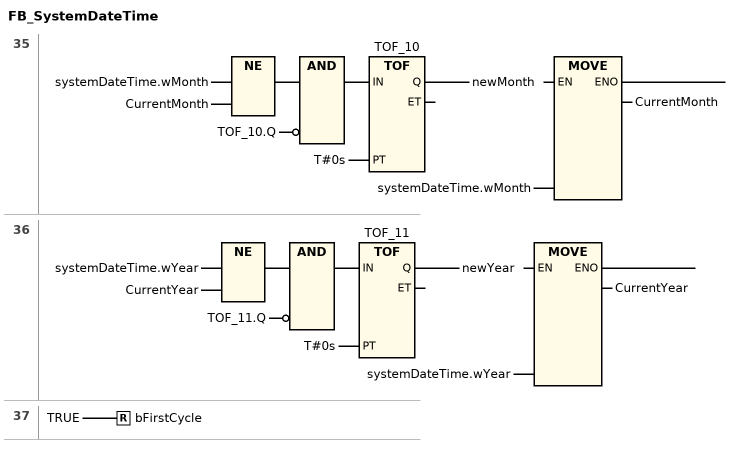
// NETWORK 35
TOF_10(IN := systemDateTime.wMonth <> CurrentMonth AND NOT TOF_10.Q, PT := T#0s); // TOF
newMonth := TOF_10.Q;
IF TOF_10.Q THEN CurrentMonth := systemDateTime.wMonth; END_IF

// NETWORK 36
TOF_11(IN := systemDateTime.wYear <> CurrentYear AND NOT TOF_11.Q, PT := T#0s); // TOF
newYear := TOF_11.Q;
IF TOF_11.Q THEN CurrentYear := systemDateTime.wYear; END_IF

// NETWORK 37
bFirstCycle R= TRUE;

END_FUNCTION_BLOCK

// ---- POUs/1. Main Control/P1_00_MAIN.TcPOU
PROGRAM P1_00_MAIN
VAR
END_VAR

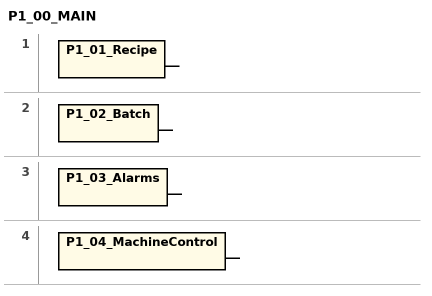
// NETWORK 1
P1_01_Recipe();

// NETWORK 2
P1_02_Batch();

// NETWORK 3
P1_03_Alarms();

// NETWORK 4
P1_04_MachineControl();

END_PROGRAM

// ---- POUs/1. Main Control/P1_01_Recipe.TcPOU
PROGRAM P1_01_Recipe
VAR
	i						:INT;
END_VAR

Recipes.Production.stPhase[1].bEnable := TRUE;
Recipes.Production_Phase_HMI.bEnable := TRUE;

Recipes.Production.iActivePhase := 0;

FOR i := 1 TO 20 DO
	IF Recipes.Production.stPhase[i].bEnable THEN
		Recipes.Production.iActivePhase := i;
	END_IF
	
	IF NOT Recipes.Production.stPhase[i].bEnable THEN
		Recipes.Production.stPhase[i] := Recipes.Production_Empty.stPhase[0];
	END_IF
END_FOR

END_PROGRAM

// ---- POUs/1. Main Control/P1_02_Batch.TcPOU
PROGRAM P1_02_Batch
VAR
	fbBatch					:FB_Batch;
	fbBatchLog				:FB_BatchLog;
END_VAR
VAR // added by the converter: edge detectors and wires of the graphical bodies
    _rt1, _rt2, _rt3 : R_TRIG;
END_VAR

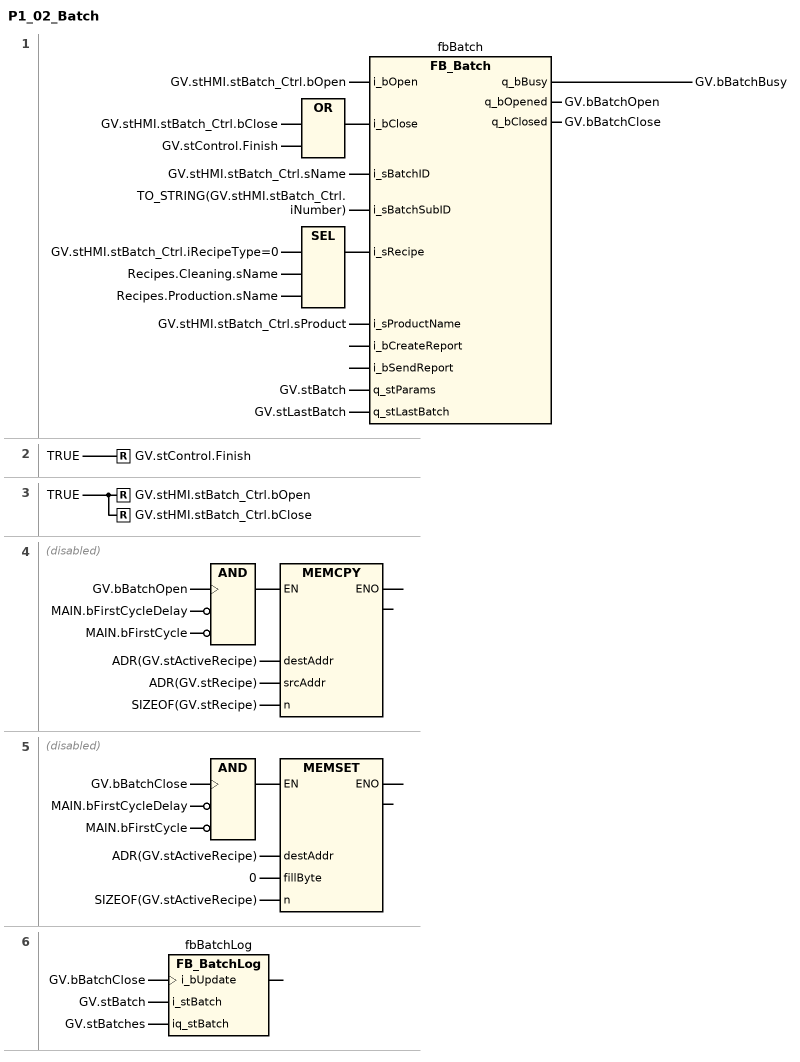
// NETWORK 1
fbBatch(
    i_bOpen := GV.stHMI.stBatch_Ctrl.bOpen,
    i_bClose := GV.stHMI.stBatch_Ctrl.bClose OR GV.stControl.Finish,
    i_sBatchID := GV.stHMI.stBatch_Ctrl.sName,
    i_sBatchSubID := TO_STRING(GV.stHMI.stBatch_Ctrl.iNumber),
    i_sRecipe := SEL(GV.stHMI.stBatch_Ctrl.iRecipeType=0, Recipes.Cleaning.sName, Recipes.Production.sName),
    i_sProductName := GV.stHMI.stBatch_Ctrl.sProduct,
    q_stParams := GV.stBatch,
    q_stLastBatch := GV.stLastBatch,
    q_bOpened => GV.bBatchOpen,
    q_bClosed => GV.bBatchClose); // FB_Batch
GV.bBatchBusy := fbBatch.q_bBusy;

// NETWORK 2
GV.stControl.Finish R= TRUE;

// NETWORK 3
GV.stHMI.stBatch_Ctrl.bOpen R= TRUE;
GV.stHMI.stBatch_Ctrl.bClose R= TRUE;

// NETWORK 4 (disabled)
// _rt1(CLK := GV.bBatchOpen);
// IF _rt1.Q AND NOT MAIN.bFirstCycleDelay AND NOT MAIN.bFirstCycle THEN
//     MEMCPY(destAddr := ADR(GV.stActiveRecipe), srcAddr := ADR(GV.stRecipe), n := SIZEOF(GV.stRecipe));
// END_IF

// NETWORK 5 (disabled)
// _rt2(CLK := GV.bBatchClose);
// IF _rt2.Q AND NOT MAIN.bFirstCycleDelay AND NOT MAIN.bFirstCycle THEN
//     MEMSET(destAddr := ADR(GV.stActiveRecipe), fillByte := 0, n := SIZEOF(GV.stActiveRecipe));
// END_IF

// NETWORK 6
_rt3(CLK := GV.bBatchClose);
fbBatchLog(i_bUpdate := _rt3.Q, i_stBatch := GV.stBatch, iq_stBatch := GV.stBatches); // FB_BatchLog

END_PROGRAM

// ---- FB/FB_Batch.TcPOU
FUNCTION_BLOCK FB_Batch
VAR_INPUT
	i_bOpen						:BOOL; 
	i_bClose					:BOOL; 
	i_iRecipeType				:INT;
	i_sBatchID					:STRING; 
	i_sBatchSubID				:STRING;
	i_sRecipe					:STRING;
	i_sProductName				:STRING;
	i_bCreateReport				:BOOL;
	i_bSendReport				:BOOL;
END_VAR
VAR_IN_OUT
	q_stParams					:ST_Batch;
	q_stLastBatch				:ST_Batch;
END_VAR
VAR_OUTPUT
	q_bBusy						:BOOL;	
	q_bOpened					:BOOL:=FALSE; 
	q_bClosed					:BOOL:=FALSE; 		
END_VAR

VAR
	tDelayCreateReport			:TON;
	tDelaySendReport			:TON;
END_VAR	

VAR PERSISTENT
	iStep						:INT;
	sUserOpened					:STRING;
END_VAR

tDelayCreateReport(IN:=(iStep=200),PT:=T#3S);
tDelaySendReport(IN:=(iStep=300),PT:=T#3S);

CASE iStep OF

	0: 
		MEMSET(ADR(q_stParams),0,SIZEOF(q_stParams));
		IF i_bOpen THEN
			iStep:=50;
		END_IF
		
	50:
		q_stParams.sRecipeType:=SEL(i_iRecipeType=0,'Cleaning','Production');
		IF i_sBatchSubID <> '0' THEN
			q_stParams.sBatchNumber:=CONCAT(i_sBatchID,'-');
			q_stParams.sBatchNumber:=CONCAT(q_stParams.sBatchNumber,i_sBatchSubID);
		ELSE
			q_stParams.sBatchNumber:=i_sBatchID;
		END_IF
		q_stParams.sRecipeName:=i_sRecipe;
		q_stParams.sProductName:=i_sProductName;
		q_stParams.sUser:=GV.sUserLogged;
		q_stParams.sStarted:=GV.stTime.sDateTime;
		sUserOpened:=GV.sUserLogged;
		iStep:=100;
			
	100:
		q_stParams.sUser:=sUserOpened;
		IF i_bClose THEN
			q_stParams.sFinished:=GV.stTime.sDateTime;
			q_stLastBatch:=q_stParams;
			iStep:=200;
		END_IF
		
	200:
		IF tDelayCreateReport.Q AND NOT i_bCreateReport THEN
			iStep:=300;
		END_IF
	300:
		IF tDelaySendReport.Q AND NOT i_bSendReport THEN
			iStep:=1000;
		END_IF
		
	1000:
		iStep:=0;	
END_CASE

q_bBusy:=iStep<>0;
q_bOpened:=iStep=100;
q_bClosed:=iStep>100;

END_FUNCTION_BLOCK

// ---- FB/FB_BatchLog.TcPOU
FUNCTION_BLOCK FB_BatchLog
VAR_INPUT
	i_bUpdate			:BOOL;
	i_stBatch			:ST_Batch;
END_VAR
VAR_IN_OUT
	iq_stBatch			:ARRAY[0..9] OF ST_Batch;
END_VAR
VAR
	i				:USINT;
	j				:USINT;
	bInsert			:BOOL;
END_VAR

IF i_bUpdate THEN
	bInsert:=FALSE;
	FOR i:=0 TO 9 DO
		IF iq_stBatch[i].sBatchNumber = '' THEN
			iq_stBatch[i]:=i_stBatch;
			bInsert:=TRUE;
			EXIT;
		END_IF
	END_FOR
	
	IF NOT bInsert THEN
		FOR j:=1 TO 9 DO
			iq_stBatch[j-1]:=iq_stBatch[j];
		END_FOR
		iq_stBatch[9]:=i_stBatch;
	END_IF
END_IF

END_FUNCTION_BLOCK

// ---- POUs/1. Main Control/P1_03_Alarms.TcPOU
PROGRAM P1_03_Alarms
VAR
	iActive				:INT;
	iAck				:INT;
	iRaise				:INT;
	
	bAlarmActive		:BOOL;
	bWarningActive		:BOOL;
	
	bAckAll				:BOOL;

	TON_Ack				:TON;
	TON_AlarmOK			:TON;

	TON_Alarm			:ARRAY[0..39] OF TON;
	
	
	
	
	Simulation	:BOOL;
	bTest: BOOL;
END_VAR
VAR // added by the converter: edge detectors and wires of the graphical bodies
    _rt1, _rt2, _rt3 : R_TRIG;
END_VAR

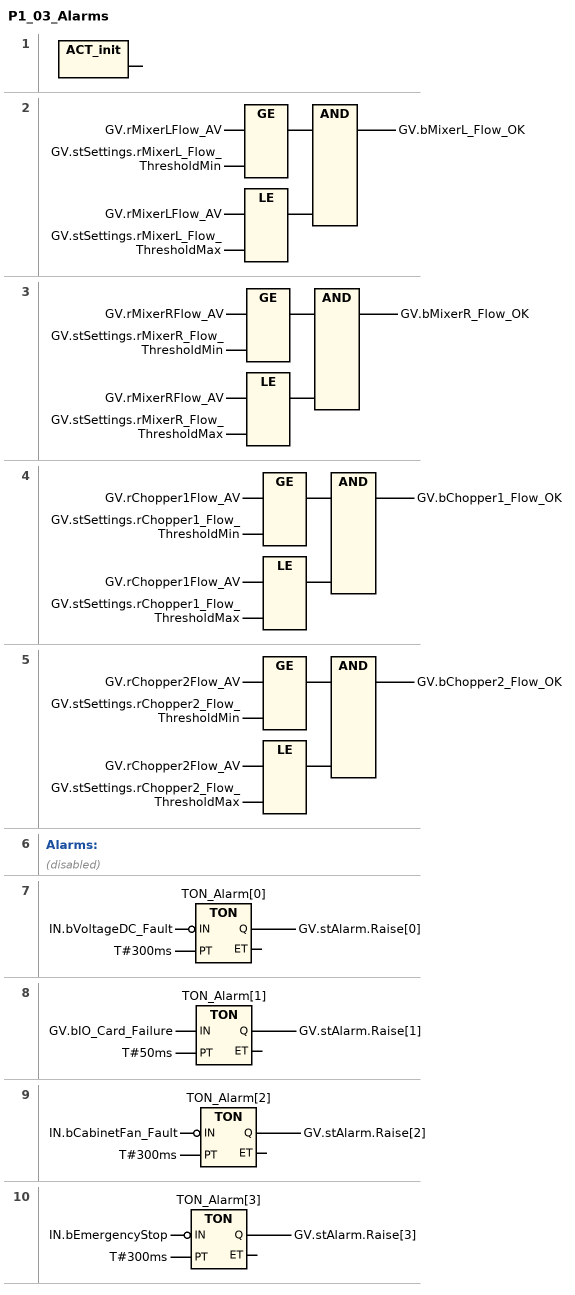
// NETWORK 1
ACT_init();

// NETWORK 2
GV.bMixerL_Flow_OK := GV.rMixerLFlow_AV >= GV.stSettings.rMixerL_Flow_ThresholdMin AND GV.rMixerLFlow_AV <= GV.stSettings.rMixerL_Flow_ThresholdMax;

// NETWORK 3
GV.bMixerR_Flow_OK := GV.rMixerRFlow_AV >= GV.stSettings.rMixerR_Flow_ThresholdMin AND GV.rMixerRFlow_AV <= GV.stSettings.rMixerR_Flow_ThresholdMax;

// NETWORK 4
GV.bChopper1_Flow_OK := GV.rChopper1Flow_AV >= GV.stSettings.rChopper1_Flow_ThresholdMin AND GV.rChopper1Flow_AV <= GV.stSettings.rChopper1_Flow_ThresholdMax;

// NETWORK 5
GV.bChopper2_Flow_OK := GV.rChopper2Flow_AV >= GV.stSettings.rChopper2_Flow_ThresholdMin AND GV.rChopper2Flow_AV <= GV.stSettings.rChopper2_Flow_ThresholdMax;

// NETWORK 6 (disabled)
// label: Alarms

// NETWORK 7
TON_Alarm[0](IN := NOT IN.bVoltageDC_Fault, PT := T#300ms); // TON
GV.stAlarm.Raise[0] := TON_Alarm[0].Q;

// NETWORK 8
TON_Alarm[1](IN := GV.bIO_Card_Failure, PT := T#50ms); // TON
GV.stAlarm.Raise[1] := TON_Alarm[1].Q;

// NETWORK 9
TON_Alarm[2](IN := NOT IN.bCabinetFan_Fault, PT := T#300ms); // TON
GV.stAlarm.Raise[2] := TON_Alarm[2].Q;

// NETWORK 10
TON_Alarm[3](IN := NOT IN.bEmergencyStop, PT := T#300ms); // TON
GV.stAlarm.Raise[3] := TON_Alarm[3].Q;

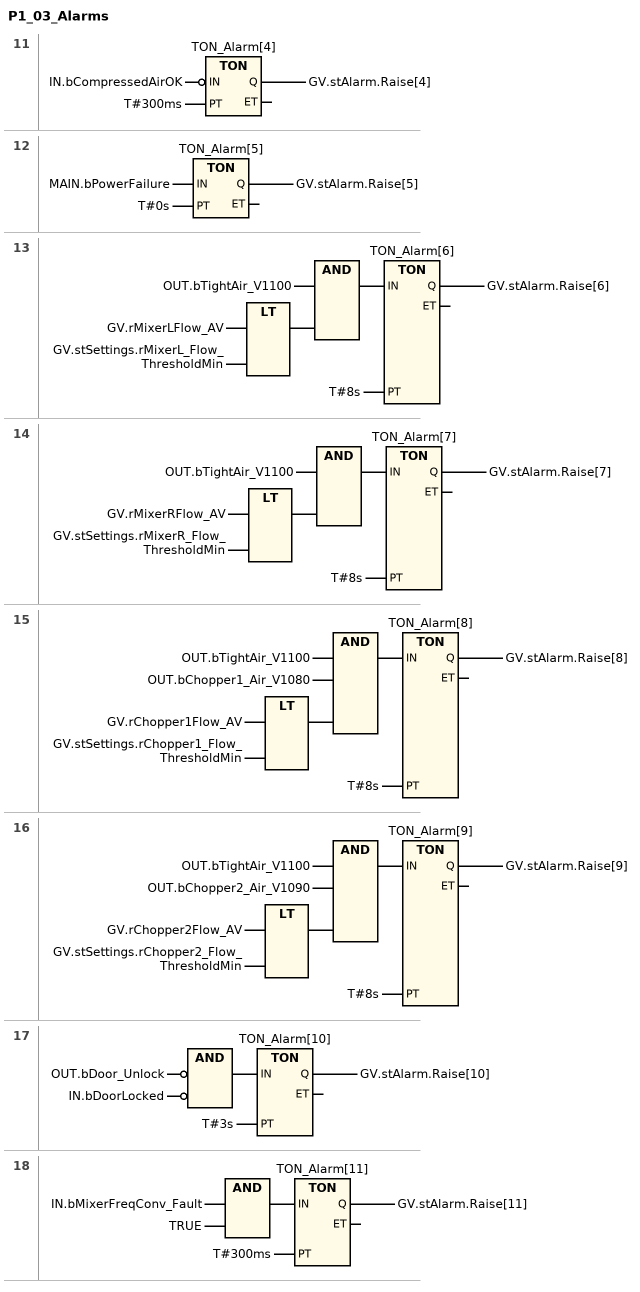
// NETWORK 11
TON_Alarm[4](IN := NOT IN.bCompressedAirOK, PT := T#300ms); // TON
GV.stAlarm.Raise[4] := TON_Alarm[4].Q;

// NETWORK 12
TON_Alarm[5](IN := MAIN.bPowerFailure, PT := T#0s); // TON
GV.stAlarm.Raise[5] := TON_Alarm[5].Q;

// NETWORK 13
TON_Alarm[6](IN := OUT.bTightAir_V1100 AND GV.rMixerLFlow_AV < GV.stSettings.rMixerL_Flow_ThresholdMin, PT := T#8s); // TON
GV.stAlarm.Raise[6] := TON_Alarm[6].Q;

// NETWORK 14
TON_Alarm[7](IN := OUT.bTightAir_V1100 AND GV.rMixerRFlow_AV < GV.stSettings.rMixerR_Flow_ThresholdMin, PT := T#8s); // TON
GV.stAlarm.Raise[7] := TON_Alarm[7].Q;

// NETWORK 15
TON_Alarm[8](IN := OUT.bTightAir_V1100 AND OUT.bChopper1_Air_V1080 AND GV.rChopper1Flow_AV < GV.stSettings.rChopper1_Flow_ThresholdMin, PT := T#8s); // TON
GV.stAlarm.Raise[8] := TON_Alarm[8].Q;

// NETWORK 16
TON_Alarm[9](IN := OUT.bTightAir_V1100 AND OUT.bChopper2_Air_V1090 AND GV.rChopper2Flow_AV < GV.stSettings.rChopper2_Flow_ThresholdMin, PT := T#8s); // TON
GV.stAlarm.Raise[9] := TON_Alarm[9].Q;

// NETWORK 17
TON_Alarm[10](IN := NOT OUT.bDoor_Unlock AND NOT IN.bDoorLocked, PT := T#3s); // TON
GV.stAlarm.Raise[10] := TON_Alarm[10].Q;

// NETWORK 18
TON_Alarm[11](IN := IN.bMixerFreqConv_Fault AND TRUE, PT := T#300ms); // TON
GV.stAlarm.Raise[11] := TON_Alarm[11].Q;

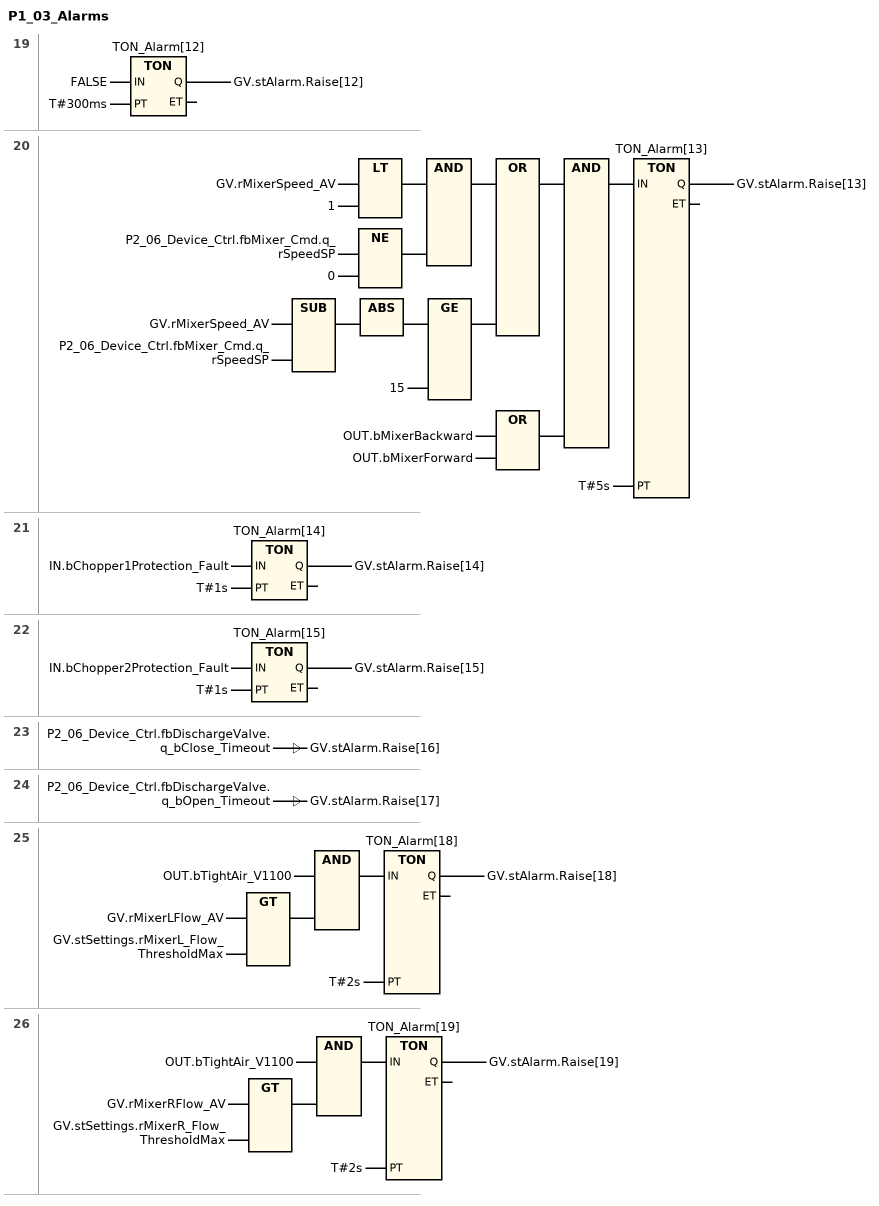
// NETWORK 19
TON_Alarm[12](IN := FALSE, PT := T#300ms); // TON
GV.stAlarm.Raise[12] := TON_Alarm[12].Q;

// NETWORK 20
TON_Alarm[13](IN := (GV.rMixerSpeed_AV < 1 AND P2_06_Device_Ctrl.fbMixer_Cmd.q_rSpeedSP <> 0 OR ABS(GV.rMixerSpeed_AV - P2_06_Device_Ctrl.fbMixer_Cmd.q_rSpeedSP) >= 15) AND (OUT.bMixerBackward OR OUT.bMixerForward), PT := T#5s); // TON
GV.stAlarm.Raise[13] := TON_Alarm[13].Q;

// NETWORK 21
TON_Alarm[14](IN := IN.bChopper1Protection_Fault, PT := T#1s); // TON
GV.stAlarm.Raise[14] := TON_Alarm[14].Q;

// NETWORK 22
TON_Alarm[15](IN := IN.bChopper2Protection_Fault, PT := T#1s); // TON
GV.stAlarm.Raise[15] := TON_Alarm[15].Q;

// NETWORK 23
_rt1(CLK := P2_06_Device_Ctrl.fbDischargeValve.q_bClose_Timeout);
GV.stAlarm.Raise[16] := _rt1.Q;

// NETWORK 24
_rt2(CLK := P2_06_Device_Ctrl.fbDischargeValve.q_bOpen_Timeout);
GV.stAlarm.Raise[17] := _rt2.Q;

// NETWORK 25
TON_Alarm[18](IN := OUT.bTightAir_V1100 AND GV.rMixerLFlow_AV > GV.stSettings.rMixerL_Flow_ThresholdMax, PT := T#2s); // TON
GV.stAlarm.Raise[18] := TON_Alarm[18].Q;

// NETWORK 26
TON_Alarm[19](IN := OUT.bTightAir_V1100 AND GV.rMixerRFlow_AV > GV.stSettings.rMixerR_Flow_ThresholdMax, PT := T#2s); // TON
GV.stAlarm.Raise[19] := TON_Alarm[19].Q;

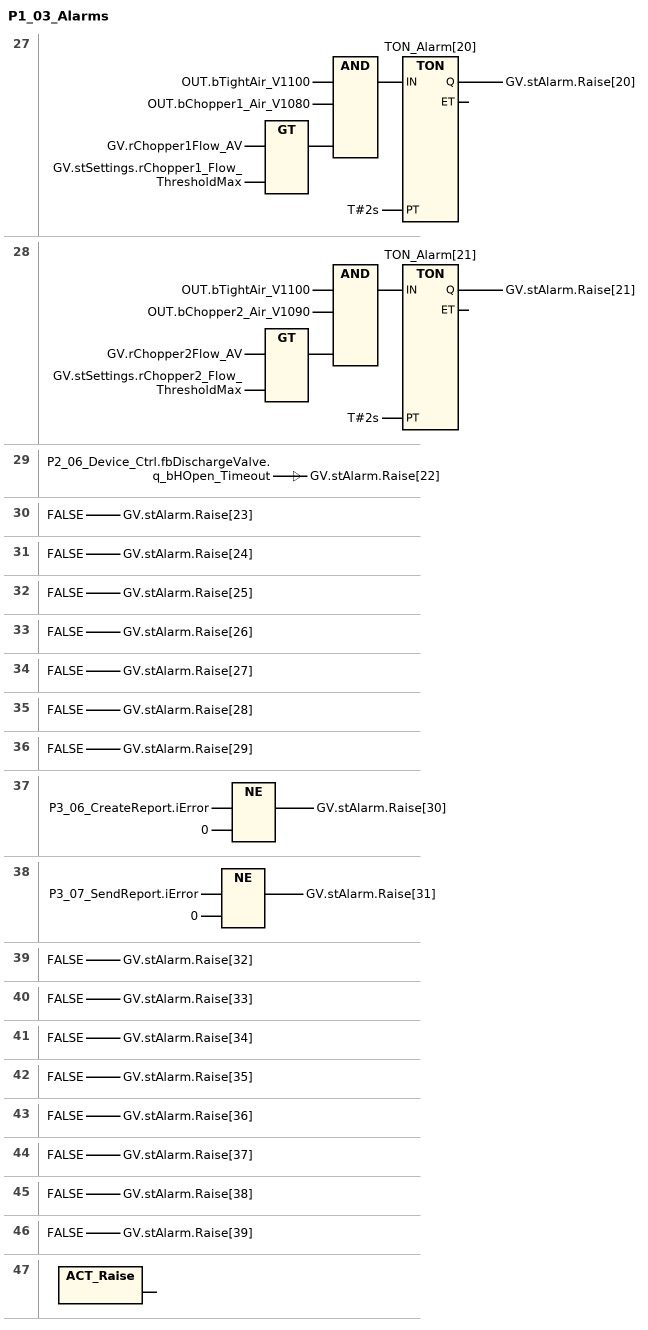
// NETWORK 27
TON_Alarm[20](IN := OUT.bTightAir_V1100 AND OUT.bChopper1_Air_V1080 AND GV.rChopper1Flow_AV > GV.stSettings.rChopper1_Flow_ThresholdMax, PT := T#2s); // TON
GV.stAlarm.Raise[20] := TON_Alarm[20].Q;

// NETWORK 28
TON_Alarm[21](IN := OUT.bTightAir_V1100 AND OUT.bChopper2_Air_V1090 AND GV.rChopper2Flow_AV > GV.stSettings.rChopper2_Flow_ThresholdMax, PT := T#2s); // TON
GV.stAlarm.Raise[21] := TON_Alarm[21].Q;

// NETWORK 29
_rt3(CLK := P2_06_Device_Ctrl.fbDischargeValve.q_bHOpen_Timeout);
GV.stAlarm.Raise[22] := _rt3.Q;

// NETWORK 30
GV.stAlarm.Raise[23] := FALSE;

// NETWORK 31
GV.stAlarm.Raise[24] := FALSE;

// NETWORK 32
GV.stAlarm.Raise[25] := FALSE;

// NETWORK 33
GV.stAlarm.Raise[26] := FALSE;

// NETWORK 34
GV.stAlarm.Raise[27] := FALSE;

// NETWORK 35
GV.stAlarm.Raise[28] := FALSE;

// NETWORK 36
GV.stAlarm.Raise[29] := FALSE;

// NETWORK 37
GV.stAlarm.Raise[30] := P3_06_CreateReport.iError <> 0;

// NETWORK 38
GV.stAlarm.Raise[31] := P3_07_SendReport.iError <> 0;

// NETWORK 39
GV.stAlarm.Raise[32] := FALSE;

// NETWORK 40
GV.stAlarm.Raise[33] := FALSE;

// NETWORK 41
GV.stAlarm.Raise[34] := FALSE;

// NETWORK 42
GV.stAlarm.Raise[35] := FALSE;

// NETWORK 43
GV.stAlarm.Raise[36] := FALSE;

// NETWORK 44
GV.stAlarm.Raise[37] := FALSE;

// NETWORK 45
GV.stAlarm.Raise[38] := FALSE;

// NETWORK 46
GV.stAlarm.Raise[39] := FALSE;

// NETWORK 47
ACT_Raise();

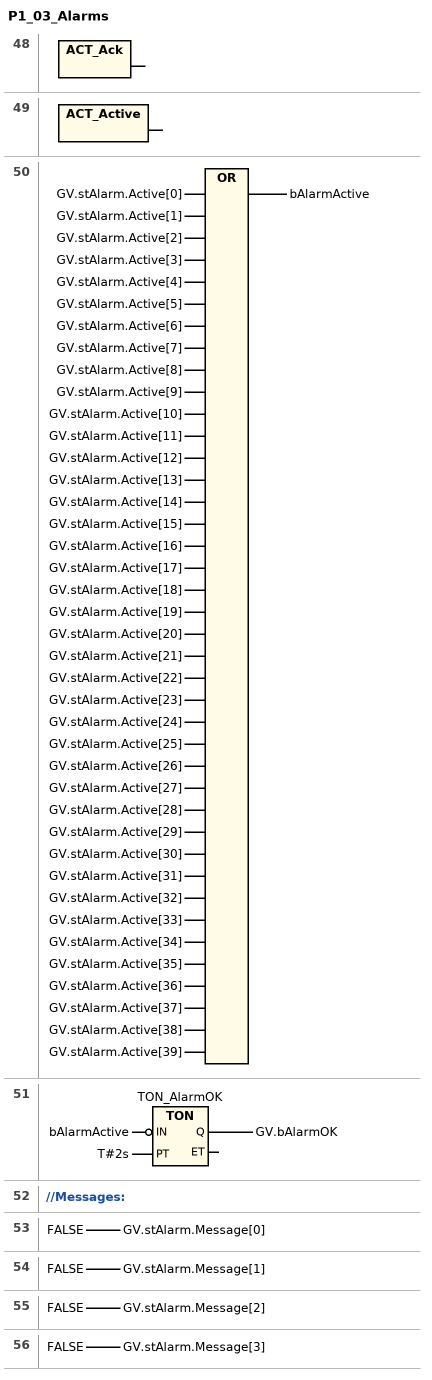
// NETWORK 48
ACT_Ack();

// NETWORK 49
ACT_Active();

// NETWORK 50
bAlarmActive := GV.stAlarm.Active[0] OR GV.stAlarm.Active[1] OR GV.stAlarm.Active[2] OR GV.stAlarm.Active[3] OR GV.stAlarm.Active[4] OR GV.stAlarm.Active[5] OR GV.stAlarm.Active[6] OR GV.stAlarm.Active[7] OR GV.stAlarm.Active[8] OR GV.stAlarm.Active[9] OR GV.stAlarm.Active[10] OR GV.stAlarm.Active[11] OR GV.stAlarm.Active[12] OR GV.stAlarm.Active[13] OR GV.stAlarm.Active[14] OR GV.stAlarm.Active[15] OR GV.stAlarm.Active[16] OR GV.stAlarm.Active[17] OR GV.stAlarm.Active[18] OR GV.stAlarm.Active[19] OR GV.stAlarm.Active[20] OR GV.stAlarm.Active[21] OR GV.stAlarm.Active[22] OR GV.stAlarm.Active[23] OR GV.stAlarm.Active[24] OR GV.stAlarm.Active[25] OR GV.stAlarm.Active[26] OR GV.stAlarm.Active[27] OR GV.stAlarm.Active[28] OR GV.stAlarm.Active[29] OR GV.stAlarm.Active[30] OR GV.stAlarm.Active[31] OR GV.stAlarm.Active[32] OR GV.stAlarm.Active[33] OR GV.stAlarm.Active[34] OR GV.stAlarm.Active[35] OR GV.stAlarm.Active[36] OR GV.stAlarm.Active[37] OR GV.stAlarm.Active[38] OR GV.stAlarm.Active[39];

// NETWORK 51
TON_AlarmOK(IN := NOT bAlarmActive, PT := T#2s); // TON
GV.bAlarmOK := TON_AlarmOK.Q;

// NETWORK 52
// label: //Messages

// NETWORK 53
GV.stAlarm.Message[0] := FALSE;

// NETWORK 54
GV.stAlarm.Message[1] := FALSE;

// NETWORK 55
GV.stAlarm.Message[2] := FALSE;

// NETWORK 56
GV.stAlarm.Message[3] := FALSE;

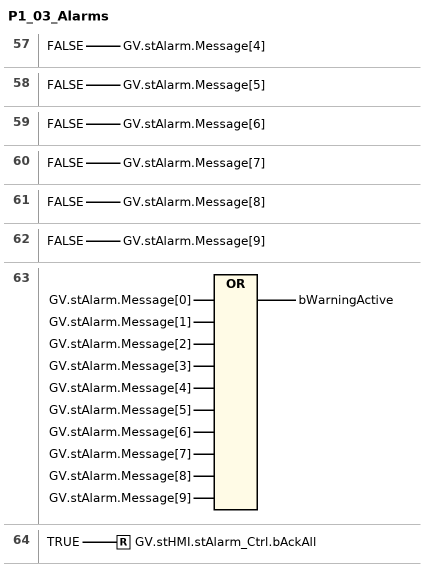
// NETWORK 57
GV.stAlarm.Message[4] := FALSE;

// NETWORK 58
GV.stAlarm.Message[5] := FALSE;

// NETWORK 59
GV.stAlarm.Message[6] := FALSE;

// NETWORK 60
GV.stAlarm.Message[7] := FALSE;

// NETWORK 61
GV.stAlarm.Message[8] := FALSE;

// NETWORK 62
GV.stAlarm.Message[9] := FALSE;

// NETWORK 63
bWarningActive := GV.stAlarm.Message[0] OR GV.stAlarm.Message[1] OR GV.stAlarm.Message[2] OR GV.stAlarm.Message[3] OR GV.stAlarm.Message[4] OR GV.stAlarm.Message[5] OR GV.stAlarm.Message[6] OR GV.stAlarm.Message[7] OR GV.stAlarm.Message[8] OR GV.stAlarm.Message[9];

// NETWORK 64
GV.stHMI.stAlarm_Ctrl.bAckAll R= TRUE;

ACTION ACT_Ack:
FOR iAck:=0 TO 99 DO
	IF GV.stAlarm.Alarm[iAck].eConfirmationState = 3 OR GV.stHMI.stAlarm_Ctrl.bAckAll THEN
		GV.stAlarm.Alarm[iAck].Clear(0,1);
	END_IF
	
	IF GV.stAlarm.Warning[iAck].bRaised AND NOT GV.stAlarm.Message[iAck] THEN
		GV.stAlarm.Warning[iAck].Clear(0,1);
	END_IF
END_FOR
END_ACTION

ACTION ACT_Active:
FOR iActive:=0 TO 99 DO
	GV.stAlarm.Active[iActive]:=GV.stAlarm.Alarm[iActive].bActive;
END_FOR
END_ACTION

ACTION ACT_Init:
IF MAIN.bFirstCycle THEN
	//Critical
	GV.stAlarm.Alarm[0].CreateEx(TC_EVENTS.Alarms.AlarmsEvent1,1,0);
	GV.stAlarm.Alarm[1].CreateEx(TC_EVENTS.Alarms.AlarmsEvent2,1,0);
	GV.stAlarm.Alarm[2].CreateEx(TC_EVENTS.Alarms.AlarmsEvent3,1,0);
	GV.stAlarm.Alarm[3].CreateEx(TC_EVENTS.Alarms.AlarmsEvent4,1,0);
	GV.stAlarm.Alarm[4].CreateEx(TC_EVENTS.Alarms.AlarmsEvent5,1,0);
	GV.stAlarm.Alarm[5].CreateEx(TC_EVENTS.Alarms.AlarmsEvent6,1,0);
	GV.stAlarm.Alarm[6].CreateEx(TC_EVENTS.Alarms.AlarmsEvent7,1,0);
	GV.stAlarm.Alarm[7].CreateEx(TC_EVENTS.Alarms.AlarmsEvent8,1,0);
	GV.stAlarm.Alarm[8].CreateEx(TC_EVENTS.Alarms.AlarmsEvent9,1,0);
	GV.stAlarm.Alarm[9].CreateEx(TC_EVENTS.Alarms.AlarmsEvent10,1,0);
	GV.stAlarm.Alarm[10].CreateEx(TC_EVENTS.Alarms.AlarmsEvent11,1,0);
	GV.stAlarm.Alarm[11].CreateEx(TC_EVENTS.Alarms.AlarmsEvent12,1,0);
	GV.stAlarm.Alarm[12].CreateEx(TC_EVENTS.Alarms.AlarmsEvent13,1,0);
	GV.stAlarm.Alarm[13].CreateEx(TC_EVENTS.Alarms.AlarmsEvent14,1,0);
	GV.stAlarm.Alarm[14].CreateEx(TC_EVENTS.Alarms.AlarmsEvent15,1,0);
	GV.stAlarm.Alarm[15].CreateEx(TC_EVENTS.Alarms.AlarmsEvent16,1,0);
	GV.stAlarm.Alarm[16].CreateEx(TC_EVENTS.Alarms.AlarmsEvent17,1,0);
	GV.stAlarm.Alarm[17].CreateEx(TC_EVENTS.Alarms.AlarmsEvent18,1,0);
	GV.stAlarm.Alarm[18].CreateEx(TC_EVENTS.Alarms.AlarmsEvent19,1,0);
	GV.stAlarm.Alarm[19].CreateEx(TC_EVENTS.Alarms.AlarmsEvent20,1,0);
	GV.stAlarm.Alarm[20].CreateEx(TC_EVENTS.Alarms.AlarmsEvent21,1,0);
	GV.stAlarm.Alarm[21].CreateEx(TC_EVENTS.Alarms.AlarmsEvent22,1,0);
	GV.stAlarm.Alarm[22].CreateEx(TC_EVENTS.Alarms.AlarmsEvent23,1,0);
	GV.stAlarm.Alarm[23].CreateEx(TC_EVENTS.Alarms.AlarmsEvent24,1,0);
	GV.stAlarm.Alarm[24].CreateEx(TC_EVENTS.Alarms.AlarmsEvent25,1,0);
	GV.stAlarm.Alarm[25].CreateEx(TC_EVENTS.Alarms.AlarmsEvent26,1,0);
	GV.stAlarm.Alarm[26].CreateEx(TC_EVENTS.Alarms.AlarmsEvent27,1,0);
	GV.stAlarm.Alarm[27].CreateEx(TC_EVENTS.Alarms.AlarmsEvent28,1,0);
	GV.stAlarm.Alarm[28].CreateEx(TC_EVENTS.Alarms.AlarmsEvent29,1,0);
	GV.stAlarm.Alarm[29].CreateEx(TC_EVENTS.Alarms.AlarmsEvent30,1,0);
	GV.stAlarm.Alarm[30].CreateEx(TC_EVENTS.Alarms.AlarmsEvent31,1,0);
	GV.stAlarm.Alarm[31].CreateEx(TC_EVENTS.Alarms.AlarmsEvent32,1,0);
	GV.stAlarm.Alarm[32].CreateEx(TC_EVENTS.Alarms.AlarmsEvent33,1,0);
	GV.stAlarm.Alarm[33].CreateEx(TC_EVENTS.Alarms.AlarmsEvent34,1,0);
	GV.stAlarm.Alarm[34].CreateEx(TC_EVENTS.Alarms.AlarmsEvent35,1,0);
	GV.stAlarm.Alarm[35].CreateEx(TC_EVENTS.Alarms.AlarmsEvent36,1,0);
	GV.stAlarm.Alarm[36].CreateEx(TC_EVENTS.Alarms.AlarmsEvent37,1,0);
	GV.stAlarm.Alarm[37].CreateEx(TC_EVENTS.Alarms.AlarmsEvent38,1,0);
	GV.stAlarm.Alarm[38].CreateEx(TC_EVENTS.Alarms.AlarmsEvent39,1,0);
	GV.stAlarm.Alarm[39].CreateEx(TC_EVENTS.Alarms.AlarmsEvent40,1,0);	
END_IF
END_ACTION

ACTION ACT_Raise:
FOR iRaise:=0 TO 99 DO
	IF GV.stAlarm.Raise[iRaise] THEN
		GV.stAlarm.Alarm[iRaise].Raise(0);
	END_IF
	
	IF GV.stAlarm.Message[iRaise] THEN
		GV.stAlarm.Warning[iRaise].Raise(0);
	END_IF
END_FOR
END_ACTION

END_PROGRAM

// ---- POUs/2. Process/P2_06_Device_Ctrl.TcPOU
PROGRAM P2_06_Device_Ctrl
VAR
	
	fbDischargeValve				:FB_Valve53_Ctrl;	
	bDischargeOpen					:BOOL;
	bDischargeClose					:BOOL;

	fbMixer_Cmd						:FB_Mixer_Ctrl;
	fbMixerSpeed_Cmd				:FB_AnalogOutput;
	fbMixerSpeed_Cmd2				:FB_Scale;

	fChopper1_Cmd					:FB_Chopper_Ctrl;
	fChopper2_Cmd					:FB_Chopper_Ctrl;
	
	fbWater_V1020_Cmd				:FB_Valve_Ctrl;
	fbWarmWater_Cmd					:FB_Valve_Ctrl;
	fbColdWater_Cmd					:FB_Valve_Ctrl;
	fbProcessWater_V1025_Cmd		:FB_Valve_Ctrl;
	fbCleaningAir_V1030_Cmd			:FB_Valve_Ctrl;
	fbTightAir_V1100_Cmd			:FB_Valve_Ctrl;
	
	fbChopper1_Air_V1080_Cmd		:FB_Valve_Ctrl;
	fbChopper1_Water_V1580_Cmd		:FB_Valve_Ctrl;
	fbChopper1_Drain_V1150_Cmd		:FB_Valve_Ctrl;
	
	fbChopper2_Air_V1090_Cmd		:FB_Valve_Ctrl;
	fbChopper2_Water_V1570_Cmd		:FB_Valve_Ctrl;
	fbChopper2_Drain_V1160_Cmd		:FB_Valve_Ctrl;
	
	fbDrainSocket_V1010_Cmd			:FB_Valve_Ctrl;
	
	tonChopper2Delay				:TON;
	
	test		:BOOL;
	fbMixerSpeed_Cmd3: FB_Scale;
	TON_0: TON;
	TON_1: TON;
	TON_2: TON;
END_VAR

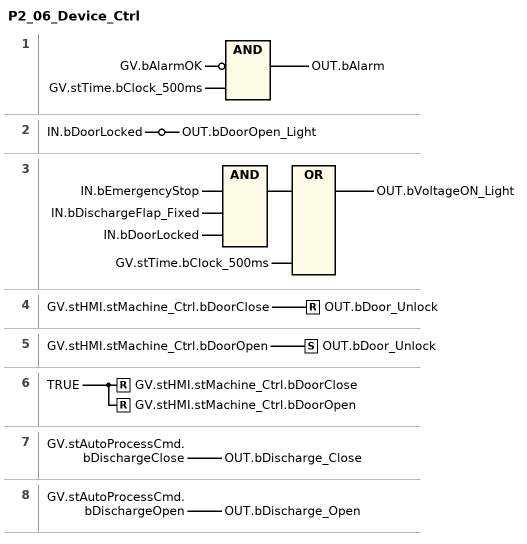
// NETWORK 1
OUT.bAlarm := NOT GV.bAlarmOK AND GV.stTime.bClock_500ms;

// NETWORK 2
OUT.bDoorOpen_Light := NOT IN.bDoorLocked;

// NETWORK 3
OUT.bVoltageON_Light := IN.bEmergencyStop AND IN.bDischargeFlap_Fixed AND IN.bDoorLocked OR GV.stTime.bClock_500ms;

// NETWORK 4
OUT.bDoor_Unlock R= GV.stHMI.stMachine_Ctrl.bDoorClose;

// NETWORK 5
OUT.bDoor_Unlock S= GV.stHMI.stMachine_Ctrl.bDoorOpen;

// NETWORK 6
GV.stHMI.stMachine_Ctrl.bDoorClose R= TRUE;
GV.stHMI.stMachine_Ctrl.bDoorOpen R= TRUE;

// NETWORK 7
OUT.bDischarge_Close := GV.stAutoProcessCmd.bDischargeClose;

// NETWORK 8
OUT.bDischarge_Open := GV.stAutoProcessCmd.bDischargeOpen;

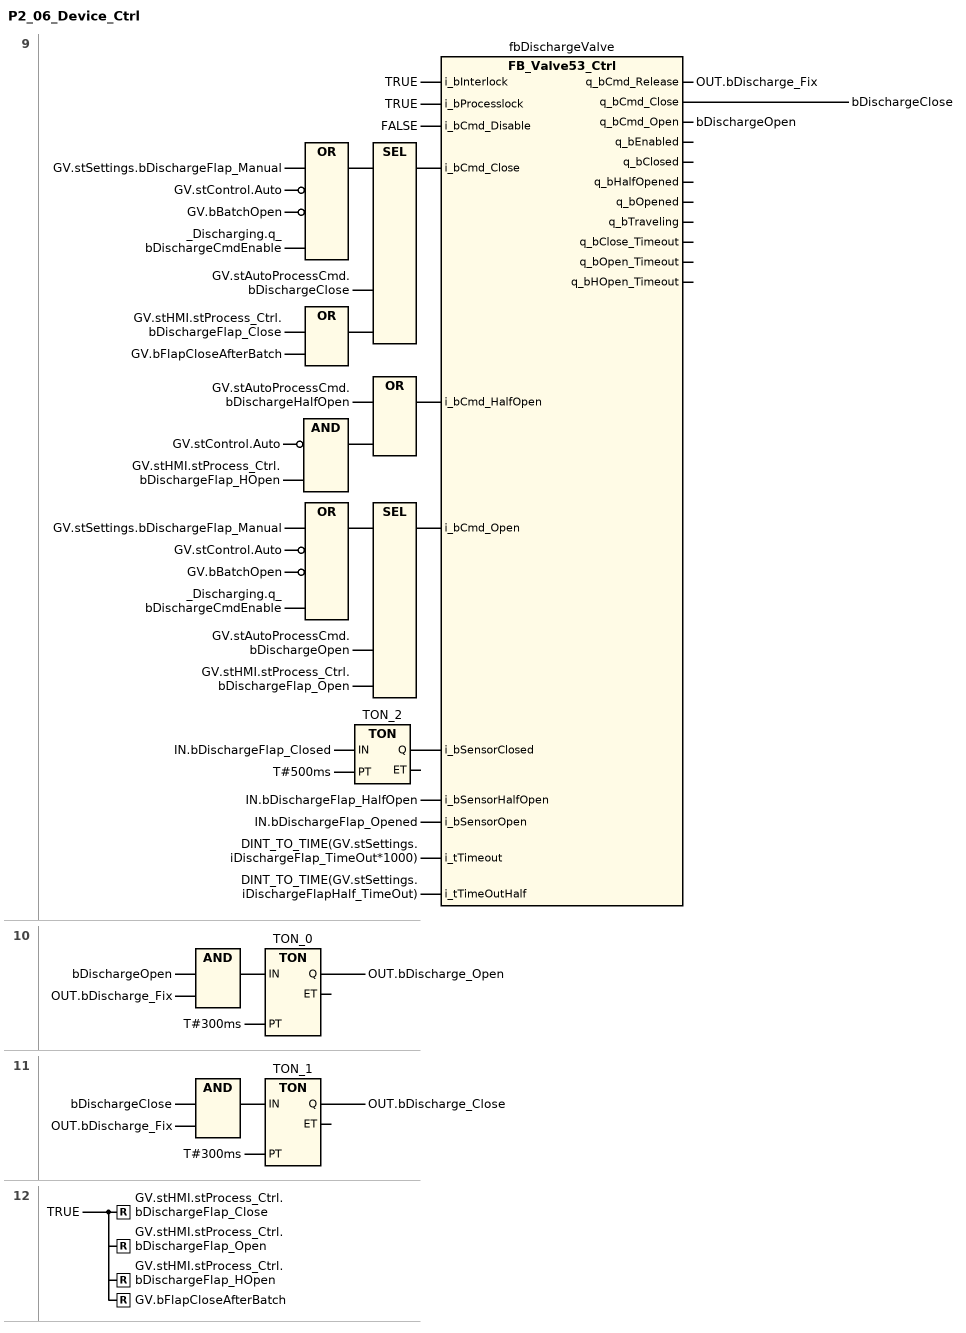
// NETWORK 9
TON_2(IN := IN.bDischargeFlap_Closed, PT := T#500ms); // TON
fbDischargeValve(
    i_bInterlock := TRUE,
    i_bProcesslock := TRUE,
    i_bCmd_Disable := FALSE,
    i_bCmd_Close := SEL(GV.stSettings.bDischargeFlap_Manual OR NOT GV.stControl.Auto OR NOT GV.bBatchOpen OR _Discharging.q_bDischargeCmdEnable, GV.stAutoProcessCmd.bDischargeClose, GV.stHMI.stProcess_Ctrl.bDischargeFlap_Close OR GV.bFlapCloseAfterBatch),
    i_bCmd_HalfOpen := GV.stAutoProcessCmd.bDischargeHalfOpen OR NOT GV.stControl.Auto AND GV.stHMI.stProcess_Ctrl.bDischargeFlap_HOpen,
    i_bCmd_Open := SEL(GV.stSettings.bDischargeFlap_Manual OR NOT GV.stControl.Auto OR NOT GV.bBatchOpen OR _Discharging.q_bDischargeCmdEnable, GV.stAutoProcessCmd.bDischargeOpen, GV.stHMI.stProcess_Ctrl.bDischargeFlap_Open),
    i_bSensorClosed := TON_2.Q,
    i_bSensorHalfOpen := IN.bDischargeFlap_HalfOpen,
    i_bSensorOpen := IN.bDischargeFlap_Opened,
    i_tTimeout := DINT_TO_TIME(GV.stSettings.iDischargeFlap_TimeOut*1000),
    i_tTimeOutHalf := DINT_TO_TIME(GV.stSettings.iDischargeFlapHalf_TimeOut),
    q_bCmd_Release => OUT.bDischarge_Fix,
    q_bCmd_Open => bDischargeOpen); // FB_Valve53_Ctrl
bDischargeClose := fbDischargeValve.q_bCmd_Close;

// NETWORK 10
TON_0(IN := bDischargeOpen AND OUT.bDischarge_Fix, PT := T#300ms); // TON
OUT.bDischarge_Open := TON_0.Q;

// NETWORK 11
TON_1(IN := bDischargeClose AND OUT.bDischarge_Fix, PT := T#300ms); // TON
OUT.bDischarge_Close := TON_1.Q;

// NETWORK 12
GV.stHMI.stProcess_Ctrl.bDischargeFlap_Close R= TRUE;
GV.stHMI.stProcess_Ctrl.bDischargeFlap_Open R= TRUE;
GV.stHMI.stProcess_Ctrl.bDischargeFlap_HOpen R= TRUE;
GV.bFlapCloseAfterBatch R= TRUE;

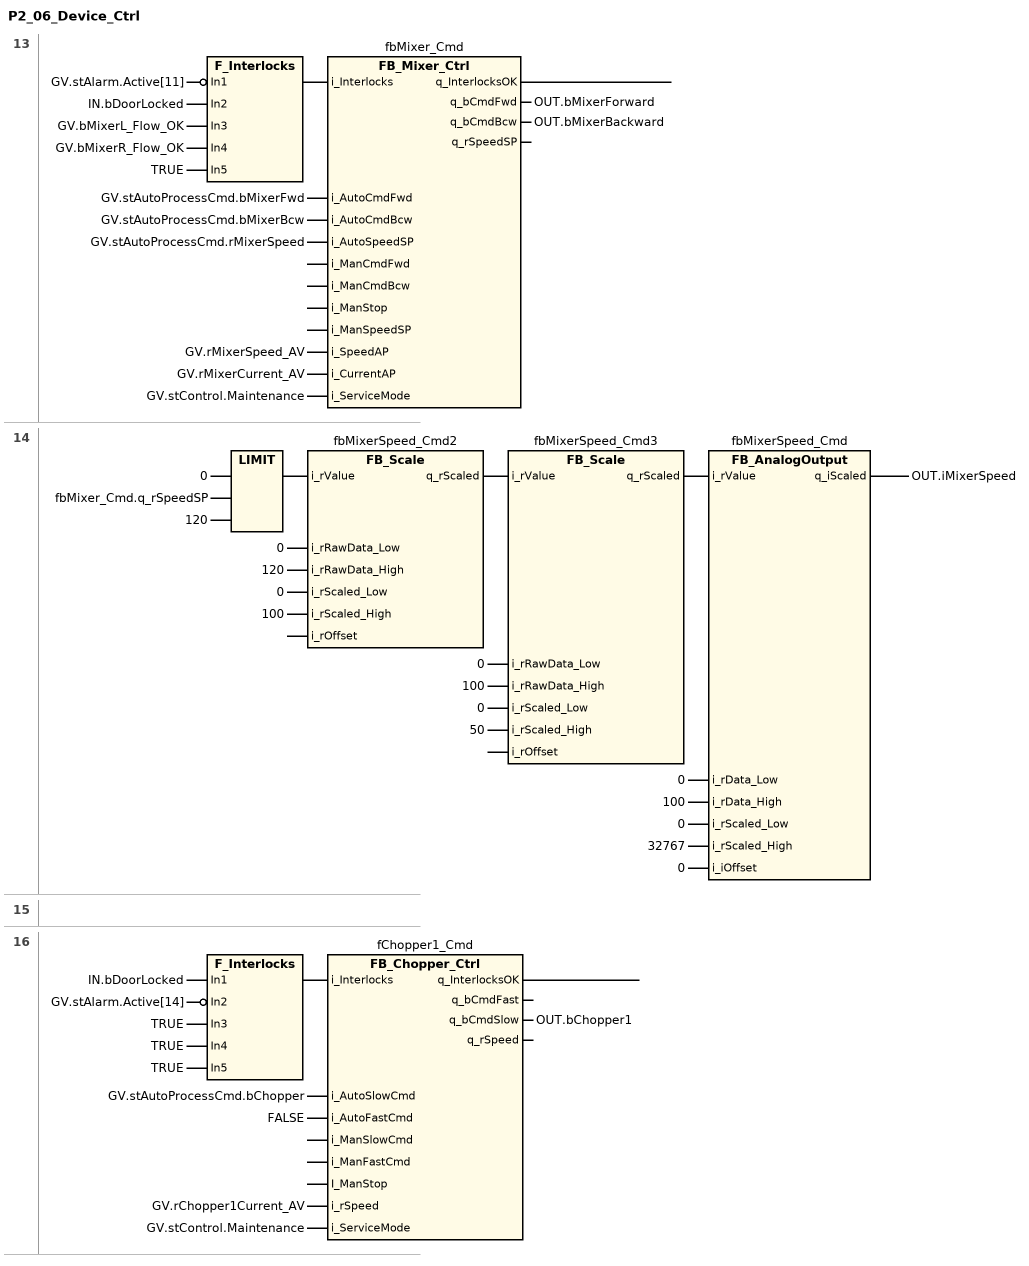
// NETWORK 13
fbMixer_Cmd(
    i_Interlocks := F_Interlocks(In1 := NOT GV.stAlarm.Active[11], In2 := IN.bDoorLocked, In3 := GV.bMixerL_Flow_OK, In4 := GV.bMixerR_Flow_OK, In5 := TRUE),
    i_AutoCmdFwd := GV.stAutoProcessCmd.bMixerFwd,
    i_AutoCmdBcw := GV.stAutoProcessCmd.bMixerBcw,
    i_AutoSpeedSP := GV.stAutoProcessCmd.rMixerSpeed,
    i_SpeedAP := GV.rMixerSpeed_AV,
    i_CurrentAP := GV.rMixerCurrent_AV,
    i_ServiceMode := GV.stControl.Maintenance,
    q_bCmdFwd => OUT.bMixerForward,
    q_bCmdBcw => OUT.bMixerBackward); // FB_Mixer_Ctrl

// NETWORK 14
fbMixerSpeed_Cmd2(
    i_rValue := LIMIT(0, fbMixer_Cmd.q_rSpeedSP, 120),
    i_rRawData_Low := 0,
    i_rRawData_High := 120,
    i_rScaled_Low := 0,
    i_rScaled_High := 100); // FB_Scale
fbMixerSpeed_Cmd3(
    i_rValue := fbMixerSpeed_Cmd2.q_rScaled,
    i_rRawData_Low := 0,
    i_rRawData_High := 100,
    i_rScaled_Low := 0,
    i_rScaled_High := 50); // FB_Scale
fbMixerSpeed_Cmd(
    i_rValue := fbMixerSpeed_Cmd3.q_rScaled,
    i_rData_Low := 0,
    i_rData_High := 100,
    i_rScaled_Low := 0,
    i_rScaled_High := 32767,
    i_iOffset := 0); // FB_AnalogOutput
OUT.iMixerSpeed := fbMixerSpeed_Cmd.q_iScaled;

// NETWORK 15

// NETWORK 16
fChopper1_Cmd(
    i_Interlocks := F_Interlocks(In1 := IN.bDoorLocked, In2 := NOT GV.stAlarm.Active[14], In3 := TRUE, In4 := TRUE, In5 := TRUE),
    i_AutoSlowCmd := GV.stAutoProcessCmd.bChopper,
    i_AutoFastCmd := FALSE,
    i_rSpeed := GV.rChopper1Current_AV,
    i_ServiceMode := GV.stControl.Maintenance,
    q_bCmdSlow => OUT.bChopper1); // FB_Chopper_Ctrl

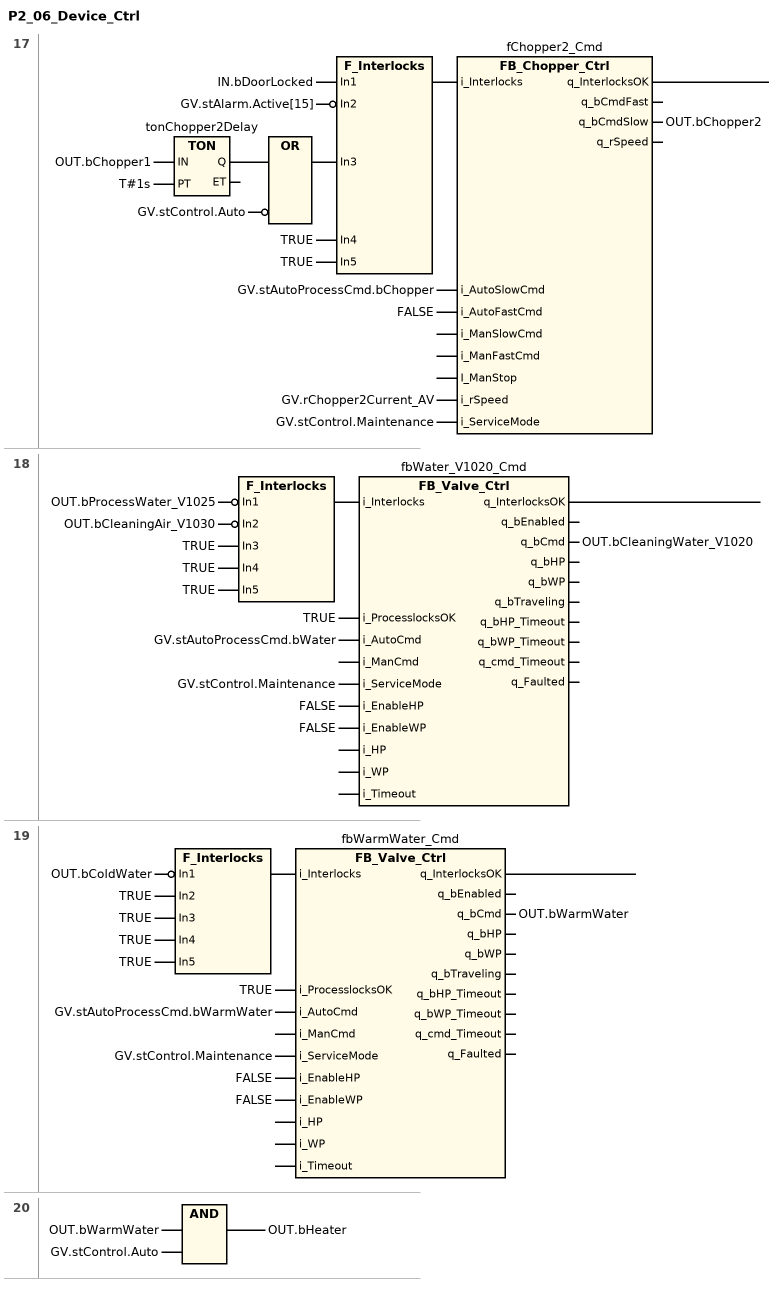
// NETWORK 17
tonChopper2Delay(IN := OUT.bChopper1, PT := T#1s); // TON
fChopper2_Cmd(
    i_Interlocks := F_Interlocks(In1 := IN.bDoorLocked, In2 := NOT GV.stAlarm.Active[15], In3 := tonChopper2Delay.Q OR NOT GV.stControl.Auto, In4 := TRUE, In5 := TRUE),
    i_AutoSlowCmd := GV.stAutoProcessCmd.bChopper,
    i_AutoFastCmd := FALSE,
    i_rSpeed := GV.rChopper2Current_AV,
    i_ServiceMode := GV.stControl.Maintenance,
    q_bCmdSlow => OUT.bChopper2); // FB_Chopper_Ctrl

// NETWORK 18
fbWater_V1020_Cmd(
    i_Interlocks := F_Interlocks(In1 := NOT OUT.bProcessWater_V1025, In2 := NOT OUT.bCleaningAir_V1030, In3 := TRUE, In4 := TRUE, In5 := TRUE),
    i_ProcesslocksOK := TRUE,
    i_AutoCmd := GV.stAutoProcessCmd.bWater,
    i_ServiceMode := GV.stControl.Maintenance,
    i_EnableHP := FALSE,
    i_EnableWP := FALSE,
    q_bCmd => OUT.bCleaningWater_V1020); // FB_Valve_Ctrl

// NETWORK 19
fbWarmWater_Cmd(
    i_Interlocks := F_Interlocks(In1 := NOT OUT.bColdWater, In2 := TRUE, In3 := TRUE, In4 := TRUE, In5 := TRUE),
    i_ProcesslocksOK := TRUE,
    i_AutoCmd := GV.stAutoProcessCmd.bWarmWater,
    i_ServiceMode := GV.stControl.Maintenance,
    i_EnableHP := FALSE,
    i_EnableWP := FALSE,
    q_bCmd => OUT.bWarmWater); // FB_Valve_Ctrl

// NETWORK 20
OUT.bHeater := OUT.bWarmWater AND GV.stControl.Auto;

